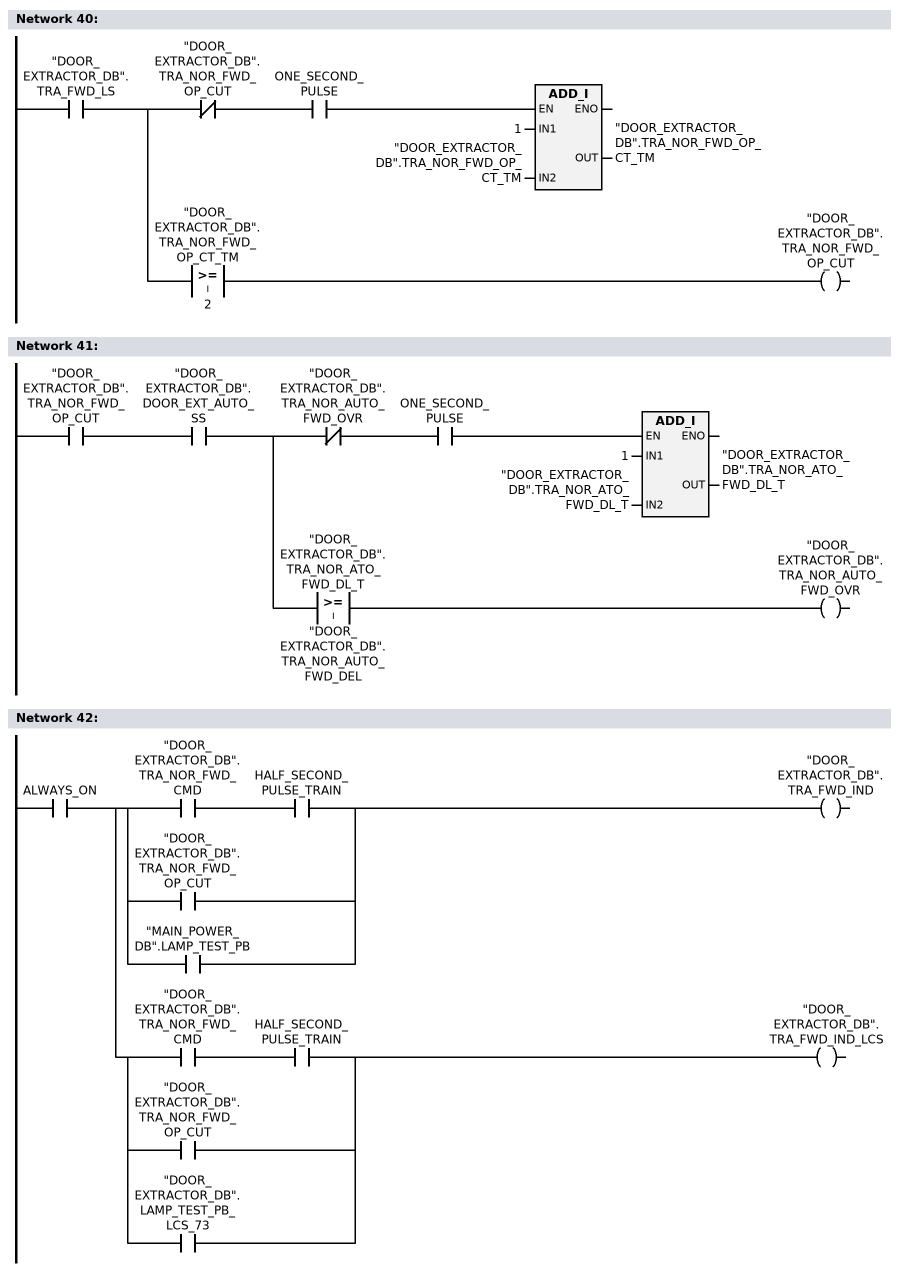
NETWORK
TITLE =
      A     "DOOR_EXTRACTOR_DB".TRA_FWD_LS;
      =     L 0.0;
      A     L 0.0;
      AN    "DOOR_EXTRACTOR_DB".TRA_NOR_FWD_OP_CUT;
      A     "ONE_SECOND_PULSE";
      JNB   M033;
      L     1;
      L     "DOOR_EXTRACTOR_DB".TRA_NOR_FWD_OP_CT_TM;
      +I;
      T     "DOOR_EXTRACTOR_DB".TRA_NOR_FWD_OP_CT_TM;
M033: NOP   0;
      A     L 0.0;
      A(;
      L     "DOOR_EXTRACTOR_DB".TRA_NOR_FWD_OP_CT_TM;
      L     2;
      >=I;
      );
      =     "DOOR_EXTRACTOR_DB".TRA_NOR_FWD_OP_CUT;
NETWORK
TITLE =
      A     "DOOR_EXTRACTOR_DB".TRA_NOR_FWD_OP_CUT;
      A     "DOOR_EXTRACTOR_DB".DOOR_EXT_AUTO_SS;
      =     L 0.0;
      A     L 0.0;
      AN    "DOOR_EXTRACTOR_DB".TRA_NOR_AUTO_FWD_OVR;
      A     "ONE_SECOND_PULSE";
      JNB   M034;
      L     1;
      L     "DOOR_EXTRACTOR_DB".TRA_NOR_ATO_FWD_DL_T;
      +I;
      T     "DOOR_EXTRACTOR_DB".TRA_NOR_ATO_FWD_DL_T;
M034: NOP   0;
      A     L 0.0;
      A(;
      L     "DOOR_EXTRACTOR_DB".TRA_NOR_ATO_FWD_DL_T;
      L     "DOOR_EXTRACTOR_DB".TRA_NOR_AUTO_FWD_DEL;
      >=I;
      );
      =     "DOOR_EXTRACTOR_DB".TRA_NOR_AUTO_FWD_OVR;
NETWORK
TITLE =
      A     "ALWAYS_ON";
      =     L 0.0;
      A     L 0.0;
      A(;
      A     "DOOR_EXTRACTOR_DB".TRA_NOR_FWD_CMD;
      A     "HALF_SECOND_PULSE_TRAIN";
      O     "DOOR_EXTRACTOR_DB".TRA_NOR_FWD_OP_CUT;
      O     "MAIN_POWER_DB".LAMP_TEST_PB;
      );
      =     "DOOR_EXTRACTOR_DB".TRA_FWD_IND;
      A     L 0.0;
      A(;
      A     "DOOR_EXTRACTOR_DB".TRA_NOR_FWD_CMD;
      A     "HALF_SECOND_PULSE_TRAIN";
      O     "DOOR_EXTRACTOR_DB".TRA_NOR_FWD_OP_CUT;
      O     "DOOR_EXTRACTOR_DB".LAMP_TEST_PB_LCS_73;
      );
      =     "DOOR_EXTRACTOR_DB".TRA_FWD_IND_LCS;
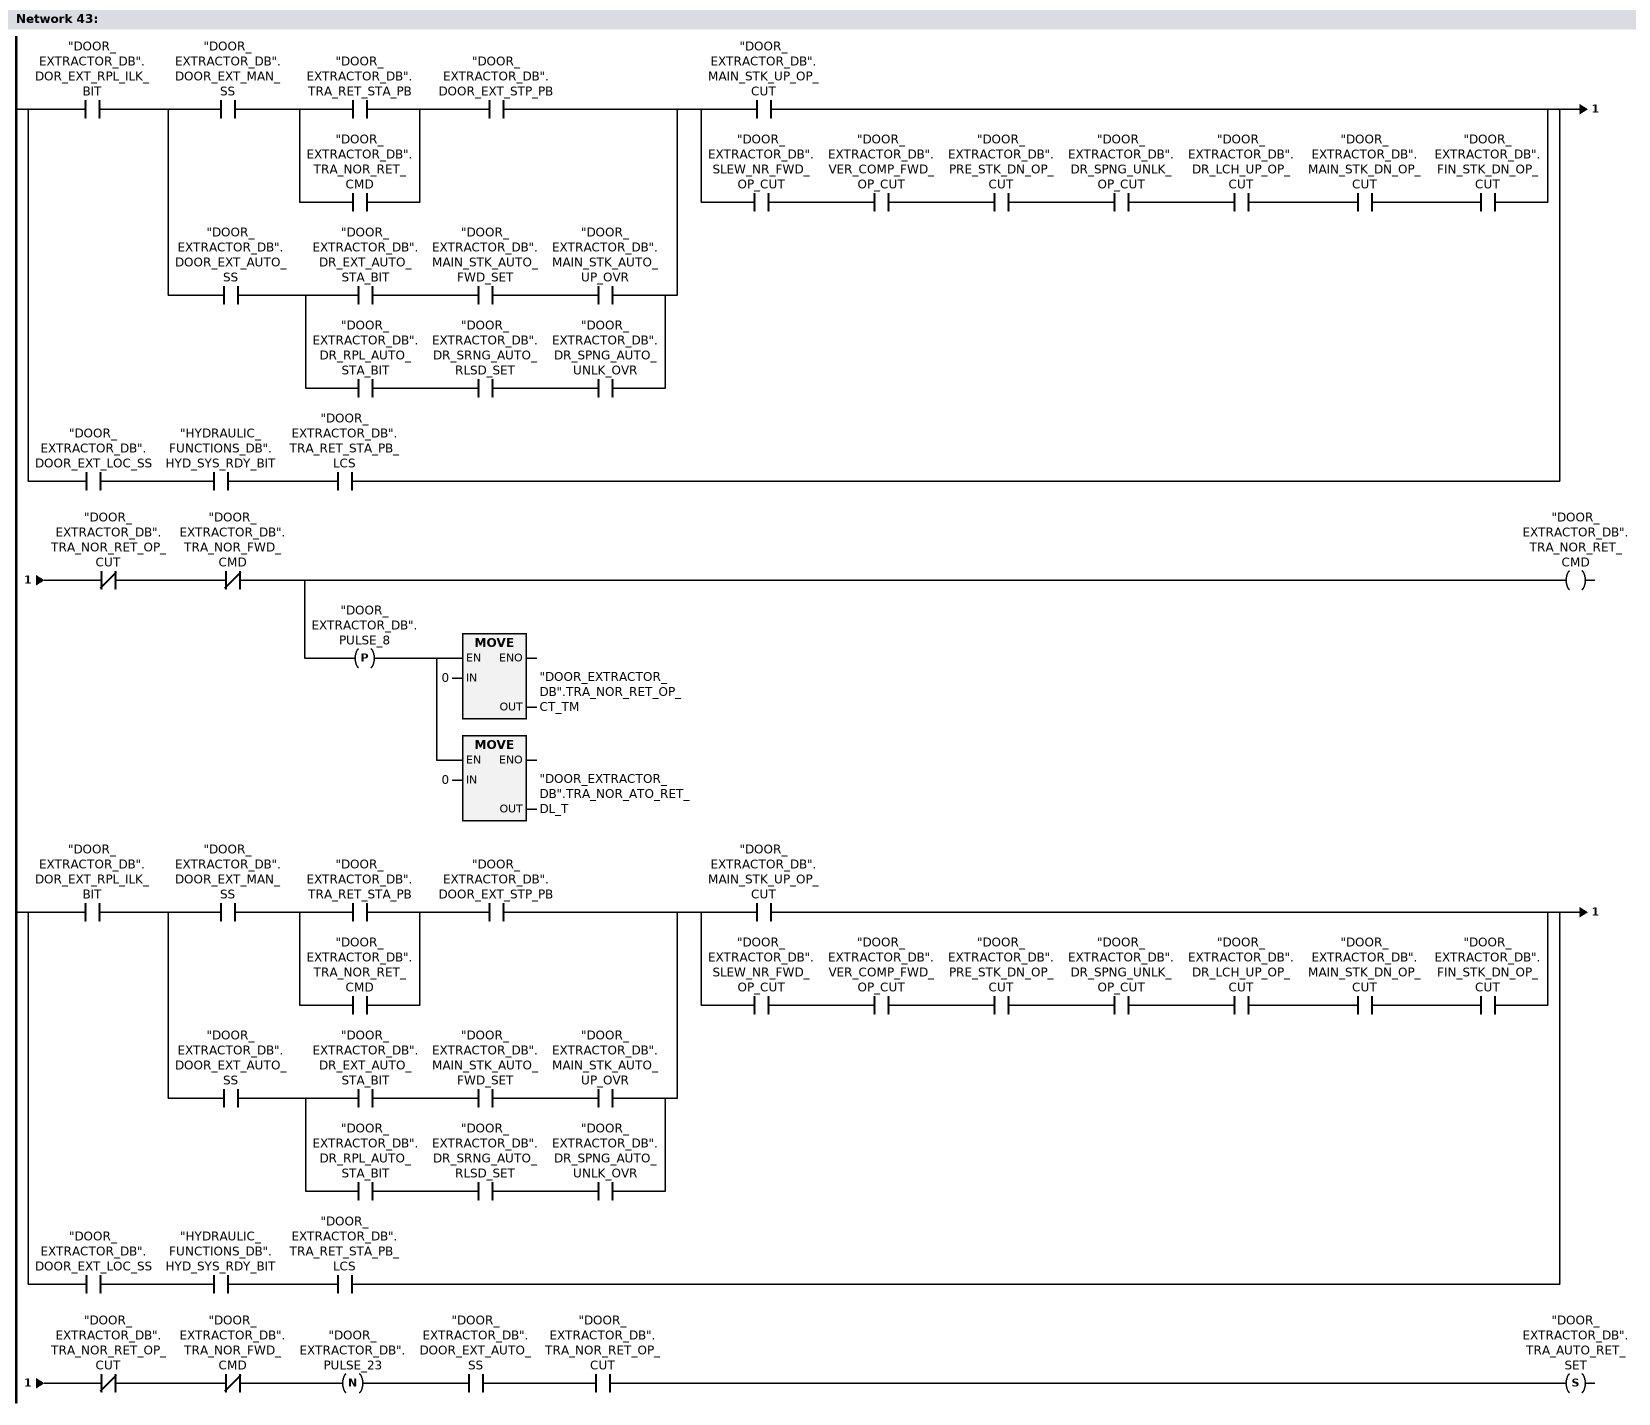
NETWORK
TITLE =
      A(;
      A     "DOOR_EXTRACTOR_DB".DOR_EXT_RPL_ILK_BIT;
      A(;
      A     "DOOR_EXTRACTOR_DB".DOOR_EXT_MAN_SS;
      A(;
      O     "DOOR_EXTRACTOR_DB".TRA_RET_STA_PB;
      O     "DOOR_EXTRACTOR_DB".TRA_NOR_RET_CMD;
      );
      A     "DOOR_EXTRACTOR_DB".DOOR_EXT_STP_PB;
      O;
      A     "DOOR_EXTRACTOR_DB".DOOR_EXT_AUTO_SS;
      A(;
      A     "DOOR_EXTRACTOR_DB".DR_EXT_AUTO_STA_BIT;
      A     "DOOR_EXTRACTOR_DB".MAIN_STK_AUTO_FWD_SET;
      A     "DOOR_EXTRACTOR_DB".MAIN_STK_AUTO_UP_OVR;
      O;
      A     "DOOR_EXTRACTOR_DB".DR_RPL_AUTO_STA_BIT;
      A     "DOOR_EXTRACTOR_DB".DR_SRNG_AUTO_RLSD_SET;
      A     "DOOR_EXTRACTOR_DB".DR_SPNG_AUTO_UNLK_OVR;
      );
      );
      A(;
      O     "DOOR_EXTRACTOR_DB".MAIN_STK_UP_OP_CUT;
      O;
      A     "DOOR_EXTRACTOR_DB".SLEW_NR_FWD_OP_CUT;
      A     "DOOR_EXTRACTOR_DB".VER_COMP_FWD_OP_CUT;
      A     "DOOR_EXTRACTOR_DB".PRE_STK_DN_OP_CUT;
      A     "DOOR_EXTRACTOR_DB".DR_SPNG_UNLK_OP_CUT;
      A     "DOOR_EXTRACTOR_DB".DR_LCH_UP_OP_CUT;
      A     "DOOR_EXTRACTOR_DB".MAIN_STK_DN_OP_CUT;
      A     "DOOR_EXTRACTOR_DB".FIN_STK_DN_OP_CUT;
      );
      O;
      A     "DOOR_EXTRACTOR_DB".DOOR_EXT_LOC_SS;
      A     "HYDRAULIC_FUNCTIONS_DB".HYD_SYS_RDY_BIT;
      A     "DOOR_EXTRACTOR_DB".TRA_RET_STA_PB_LCS;
      );
      AN    "DOOR_EXTRACTOR_DB".TRA_NOR_RET_OP_CUT;
      AN    "DOOR_EXTRACTOR_DB".TRA_NOR_FWD_CMD;
      =     L 0.0;
      A     L 0.0;
      BLD   102;
      =     "DOOR_EXTRACTOR_DB".TRA_NOR_RET_CMD;
      A(;
      A     L 0.0;
      FN    "DOOR_EXTRACTOR_DB".PULSE_23;
      );
      A     "DOOR_EXTRACTOR_DB".DOOR_EXT_AUTO_SS;
      A     "DOOR_EXTRACTOR_DB".TRA_NOR_RET_OP_CUT;
      S     "DOOR_EXTRACTOR_DB".TRA_AUTO_RET_SET;
      A     L 0.0;
      FP    "DOOR_EXTRACTOR_DB".PULSE_8;
      =     L 0.1;
      A     L 0.1;
      JNB   M035;
      L     0;
      T     "DOOR_EXTRACTOR_DB".TRA_NOR_RET_OP_CT_TM;
M035: NOP   0;
      A     L 0.1;
      JNB   M036;
      L     0;
      T     "DOOR_EXTRACTOR_DB".TRA_NOR_ATO_RET_DL_T;
M036: NOP   0;
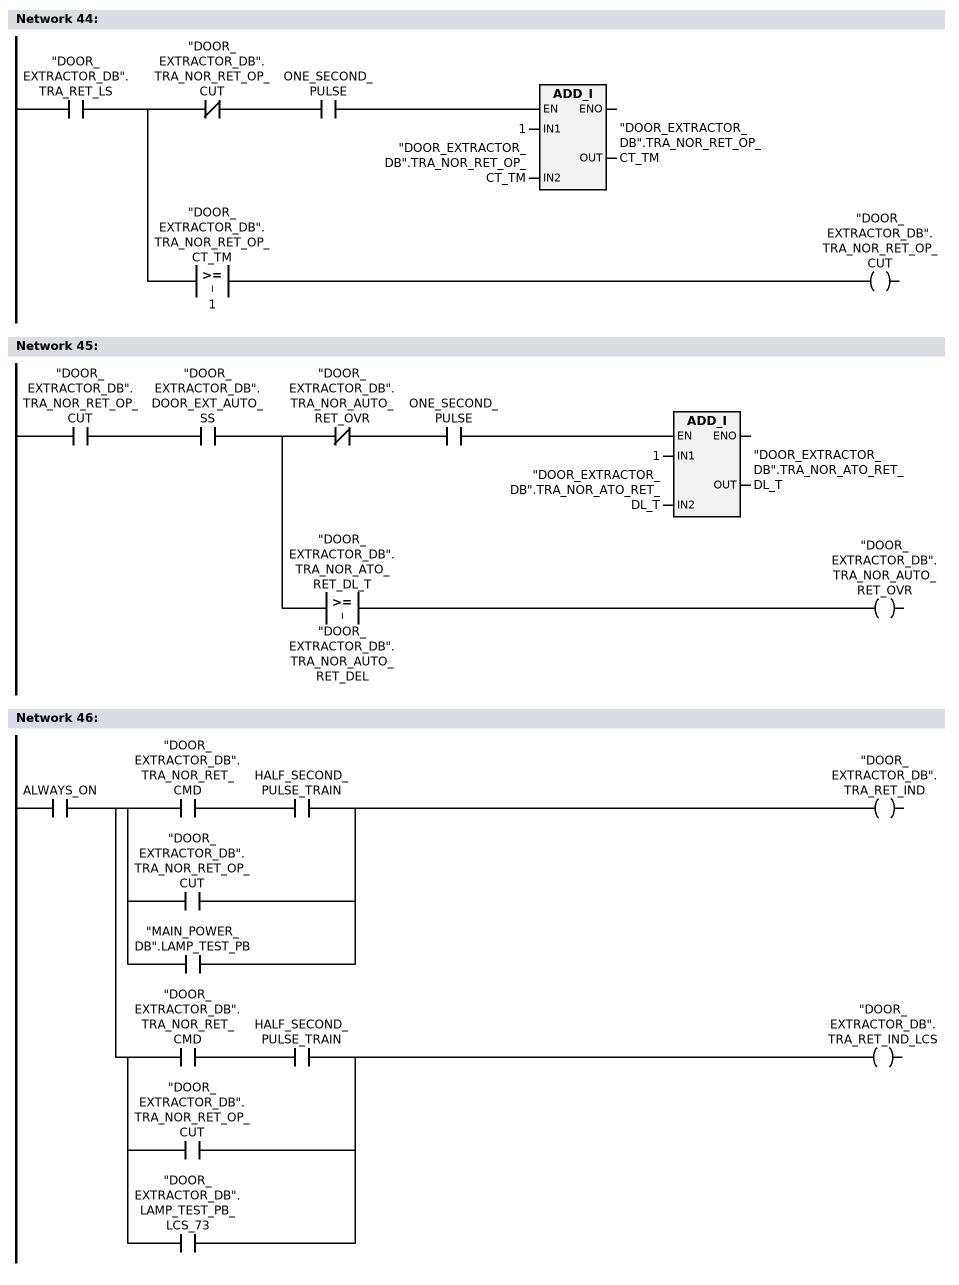
NETWORK
TITLE =
      A     "DOOR_EXTRACTOR_DB".TRA_RET_LS;
      =     L 0.0;
      A     L 0.0;
      AN    "DOOR_EXTRACTOR_DB".TRA_NOR_RET_OP_CUT;
      A     "ONE_SECOND_PULSE";
      JNB   M037;
      L     1;
      L     "DOOR_EXTRACTOR_DB".TRA_NOR_RET_OP_CT_TM;
      +I;
      T     "DOOR_EXTRACTOR_DB".TRA_NOR_RET_OP_CT_TM;
M037: NOP   0;
      A     L 0.0;
      A(;
      L     "DOOR_EXTRACTOR_DB".TRA_NOR_RET_OP_CT_TM;
      L     1;
      >=I;
      );
      =     "DOOR_EXTRACTOR_DB".TRA_NOR_RET_OP_CUT;
NETWORK
TITLE =
      A     "DOOR_EXTRACTOR_DB".TRA_NOR_RET_OP_CUT;
      A     "DOOR_EXTRACTOR_DB".DOOR_EXT_AUTO_SS;
      =     L 0.0;
      A     L 0.0;
      AN    "DOOR_EXTRACTOR_DB".TRA_NOR_AUTO_RET_OVR;
      A     "ONE_SECOND_PULSE";
      JNB   M038;
      L     1;
      L     "DOOR_EXTRACTOR_DB".TRA_NOR_ATO_RET_DL_T;
      +I;
      T     "DOOR_EXTRACTOR_DB".TRA_NOR_ATO_RET_DL_T;
M038: NOP   0;
      A     L 0.0;
      A(;
      L     "DOOR_EXTRACTOR_DB".TRA_NOR_ATO_RET_DL_T;
      L     "DOOR_EXTRACTOR_DB".TRA_NOR_AUTO_RET_DEL;
      >=I;
      );
      =     "DOOR_EXTRACTOR_DB".TRA_NOR_AUTO_RET_OVR;
NETWORK
TITLE =
      A     "ALWAYS_ON";
      =     L 0.0;
      A     L 0.0;
      A(;
      A     "DOOR_EXTRACTOR_DB".TRA_NOR_RET_CMD;
      A     "HALF_SECOND_PULSE_TRAIN";
      O     "DOOR_EXTRACTOR_DB".TRA_NOR_RET_OP_CUT;
      O     "MAIN_POWER_DB".LAMP_TEST_PB;
      );
      =     "DOOR_EXTRACTOR_DB".TRA_RET_IND;
      A     L 0.0;
      A(;
      A     "DOOR_EXTRACTOR_DB".TRA_NOR_RET_CMD;
      A     "HALF_SECOND_PULSE_TRAIN";
      O     "DOOR_EXTRACTOR_DB".TRA_NOR_RET_OP_CUT;
      O     "DOOR_EXTRACTOR_DB".LAMP_TEST_PB_LCS_73;
      );
      =     "DOOR_EXTRACTOR_DB".TRA_RET_IND_LCS;
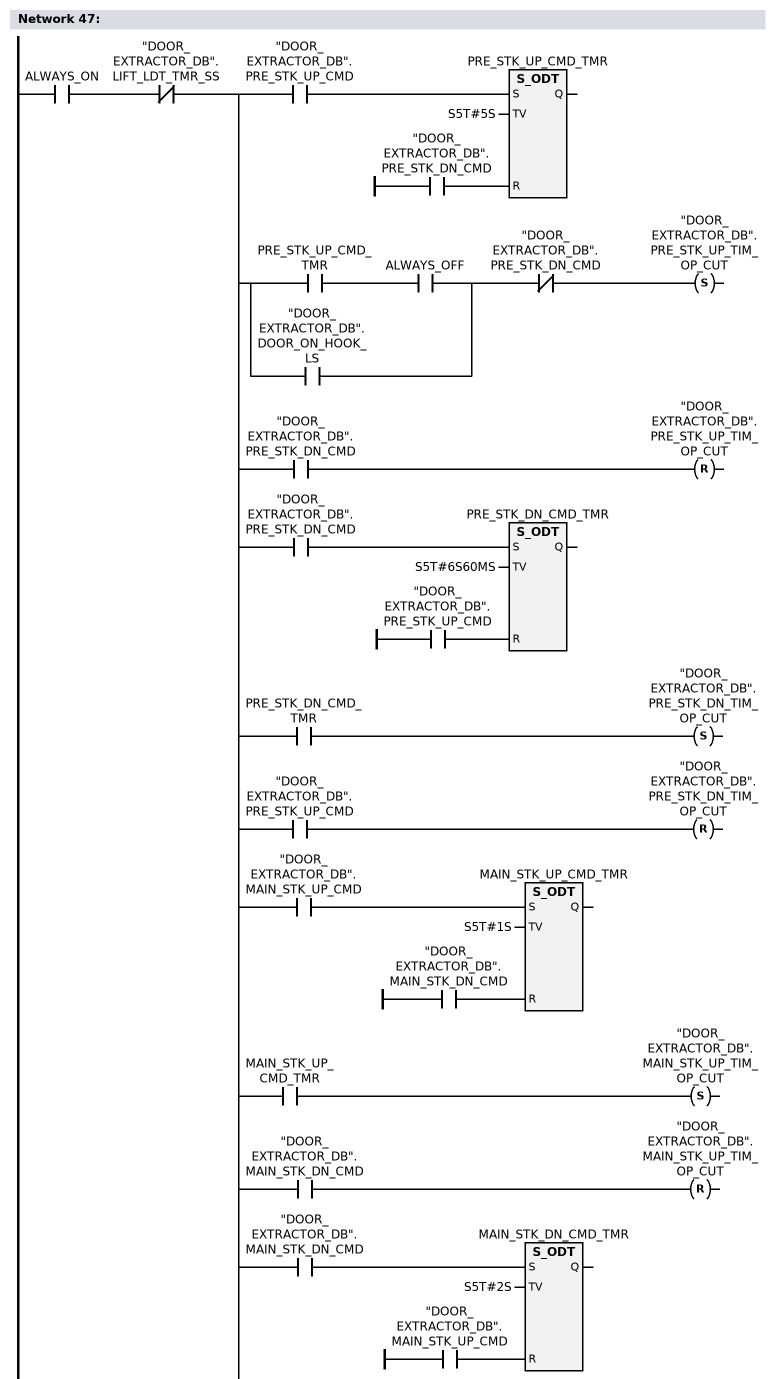
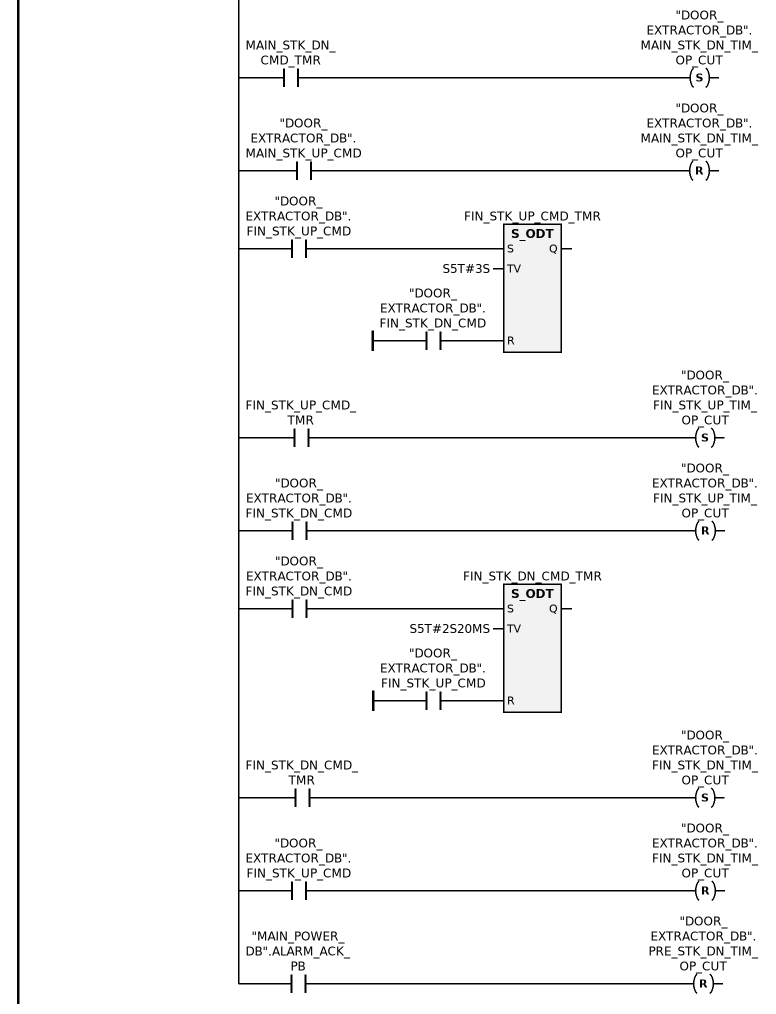
NETWORK
TITLE =
      A     "ALWAYS_ON";
      AN    "DOOR_EXTRACTOR_DB".LIFT_LDT_TMR_SS;
      =     L 0.0;
      A     L 0.0;
      A     "DOOR_EXTRACTOR_DB".PRE_STK_UP_CMD;
      L     S5T#5S;
      SD    "PRE_STK_UP_CMD_TMR";
      A     "DOOR_EXTRACTOR_DB".PRE_STK_DN_CMD;
      R     "PRE_STK_UP_CMD_TMR";
      NOP   0;
      NOP   0;
      NOP   0;
      A     L 0.0;
      A(;
      A     "PRE_STK_UP_CMD_TMR";
      A     "ALWAYS_OFF";
      O     "DOOR_EXTRACTOR_DB".DOOR_ON_HOOK_LS;
      );
      AN    "DOOR_EXTRACTOR_DB".PRE_STK_DN_CMD;
      S     "DOOR_EXTRACTOR_DB".PRE_STK_UP_TIM_OP_CUT;
      A     L 0.0;
      A     "DOOR_EXTRACTOR_DB".PRE_STK_DN_CMD;
      R     "DOOR_EXTRACTOR_DB".PRE_STK_UP_TIM_OP_CUT;
      A     L 0.0;
      A     "DOOR_EXTRACTOR_DB".PRE_STK_DN_CMD;
      L     S5T#6S60MS;
      SD    "PRE_STK_DN_CMD_TMR";
      A     "DOOR_EXTRACTOR_DB".PRE_STK_UP_CMD;
      R     "PRE_STK_DN_CMD_TMR";
      NOP   0;
      NOP   0;
      NOP   0;
      A     L 0.0;
      A     "PRE_STK_DN_CMD_TMR";
      S     "DOOR_EXTRACTOR_DB".PRE_STK_DN_TIM_OP_CUT;
      A     L 0.0;
      A     "DOOR_EXTRACTOR_DB".PRE_STK_UP_CMD;
      R     "DOOR_EXTRACTOR_DB".PRE_STK_DN_TIM_OP_CUT;
      A     L 0.0;
      A     "DOOR_EXTRACTOR_DB".MAIN_STK_UP_CMD;
      L     S5T#1S;
      SD    "MAIN_STK_UP_CMD_TMR";
      A     "DOOR_EXTRACTOR_DB".MAIN_STK_DN_CMD;
      R     "MAIN_STK_UP_CMD_TMR";
      NOP   0;
      NOP   0;
      NOP   0;
      A     L 0.0;
      A     "MAIN_STK_UP_CMD_TMR";
      S     "DOOR_EXTRACTOR_DB".MAIN_STK_UP_TIM_OP_CUT;
      A     L 0.0;
      A     "DOOR_EXTRACTOR_DB".MAIN_STK_DN_CMD;
      R     "DOOR_EXTRACTOR_DB".MAIN_STK_UP_TIM_OP_CUT;
      A     L 0.0;
      A     "DOOR_EXTRACTOR_DB".MAIN_STK_DN_CMD;
      L     S5T#2S;
      SD    "MAIN_STK_DN_CMD_TMR";
      A     "DOOR_EXTRACTOR_DB".MAIN_STK_UP_CMD;
      R     "MAIN_STK_DN_CMD_TMR";
      NOP   0;
      NOP   0;
      NOP   0;
      A     L 0.0;
      A     "MAIN_STK_DN_CMD_TMR";
      S     "DOOR_EXTRACTOR_DB".MAIN_STK_DN_TIM_OP_CUT;
      A     L 0.0;
      A     "DOOR_EXTRACTOR_DB".MAIN_STK_UP_CMD;
      R     "DOOR_EXTRACTOR_DB".MAIN_STK_DN_TIM_OP_CUT;
      A     L 0.0;
      A     "DOOR_EXTRACTOR_DB".FIN_STK_UP_CMD;
      L     S5T#3S;
      SD    "FIN_STK_UP_CMD_TMR";
      A     "DOOR_EXTRACTOR_DB".FIN_STK_DN_CMD;
      R     "FIN_STK_UP_CMD_TMR";
      NOP   0;
      NOP   0;
      NOP   0;
      A     L 0.0;
      A     "FIN_STK_UP_CMD_TMR";
      S     "DOOR_EXTRACTOR_DB".FIN_STK_UP_TIM_OP_CUT;
      A     L 0.0;
      A     "DOOR_EXTRACTOR_DB".FIN_STK_DN_CMD;
      R     "DOOR_EXTRACTOR_DB".FIN_STK_UP_TIM_OP_CUT;
      A     L 0.0;
      A     "DOOR_EXTRACTOR_DB".FIN_STK_DN_CMD;
      L     S5T#2S20MS;
      SD    "FIN_STK_DN_CMD_TMR";
      A     "DOOR_EXTRACTOR_DB".FIN_STK_UP_CMD;
      R     "FIN_STK_DN_CMD_TMR";
      NOP   0;
      NOP   0;
      NOP   0;
      A     L 0.0;
      A     "FIN_STK_DN_CMD_TMR";
      S     "DOOR_EXTRACTOR_DB".FIN_STK_DN_TIM_OP_CUT;
      A     L 0.0;
      A     "DOOR_EXTRACTOR_DB".FIN_STK_UP_CMD;
      R     "DOOR_EXTRACTOR_DB".FIN_STK_DN_TIM_OP_CUT;
      A     L 0.0;
      A     "MAIN_POWER_DB".ALARM_ACK_PB;
      R     "DOOR_EXTRACTOR_DB".PRE_STK_DN_TIM_OP_CUT;
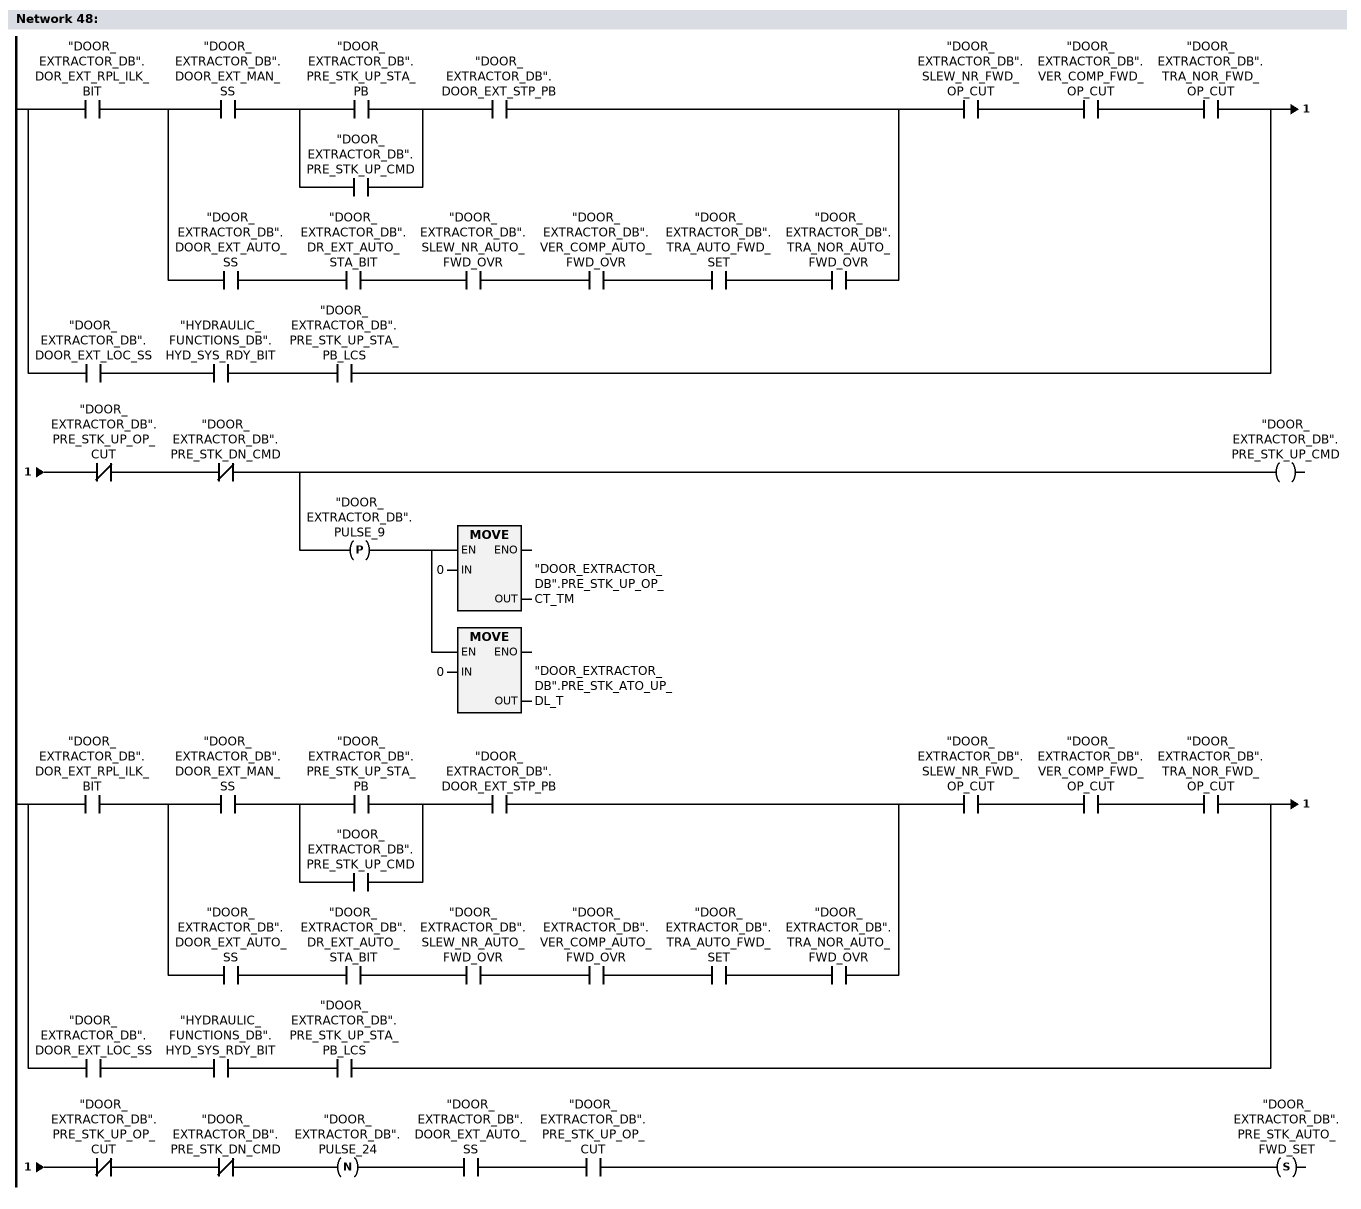
NETWORK
TITLE =
      A(;
      A     "DOOR_EXTRACTOR_DB".DOR_EXT_RPL_ILK_BIT;
      A(;
      A     "DOOR_EXTRACTOR_DB".DOOR_EXT_MAN_SS;
      A(;
      O     "DOOR_EXTRACTOR_DB".PRE_STK_UP_STA_PB;
      O     "DOOR_EXTRACTOR_DB".PRE_STK_UP_CMD;
      );
      A     "DOOR_EXTRACTOR_DB".DOOR_EXT_STP_PB;
      O;
      A     "DOOR_EXTRACTOR_DB".DOOR_EXT_AUTO_SS;
      A     "DOOR_EXTRACTOR_DB".DR_EXT_AUTO_STA_BIT;
      A     "DOOR_EXTRACTOR_DB".SLEW_NR_AUTO_FWD_OVR;
      A     "DOOR_EXTRACTOR_DB".VER_COMP_AUTO_FWD_OVR;
      A     "DOOR_EXTRACTOR_DB".TRA_AUTO_FWD_SET;
      A     "DOOR_EXTRACTOR_DB".TRA_NOR_AUTO_FWD_OVR;
      );
      A     "DOOR_EXTRACTOR_DB".SLEW_NR_FWD_OP_CUT;
      A     "DOOR_EXTRACTOR_DB".VER_COMP_FWD_OP_CUT;
      A     "DOOR_EXTRACTOR_DB".TRA_NOR_FWD_OP_CUT;
      O;
      A     "DOOR_EXTRACTOR_DB".DOOR_EXT_LOC_SS;
      A     "HYDRAULIC_FUNCTIONS_DB".HYD_SYS_RDY_BIT;
      A     "DOOR_EXTRACTOR_DB".PRE_STK_UP_STA_PB_LCS;
      );
      AN    "DOOR_EXTRACTOR_DB".PRE_STK_UP_OP_CUT;
      AN    "DOOR_EXTRACTOR_DB".PRE_STK_DN_CMD;
      =     L 0.0;
      A     L 0.0;
      BLD   102;
      =     "DOOR_EXTRACTOR_DB".PRE_STK_UP_CMD;
      A(;
      A     L 0.0;
      FN    "DOOR_EXTRACTOR_DB".PULSE_24;
      );
      A     "DOOR_EXTRACTOR_DB".DOOR_EXT_AUTO_SS;
      A     "DOOR_EXTRACTOR_DB".PRE_STK_UP_OP_CUT;
      S     "DOOR_EXTRACTOR_DB".PRE_STK_AUTO_FWD_SET;
      A     L 0.0;
      FP    "DOOR_EXTRACTOR_DB".PULSE_9;
      =     L 0.1;
      A     L 0.1;
      JNB   M039;
      L     0;
      T     "DOOR_EXTRACTOR_DB".PRE_STK_UP_OP_CT_TM;
M039: NOP   0;
      A     L 0.1;
      JNB   M040;
      L     0;
      T     "DOOR_EXTRACTOR_DB".PRE_STK_ATO_UP_DL_T;
M040: NOP   0;
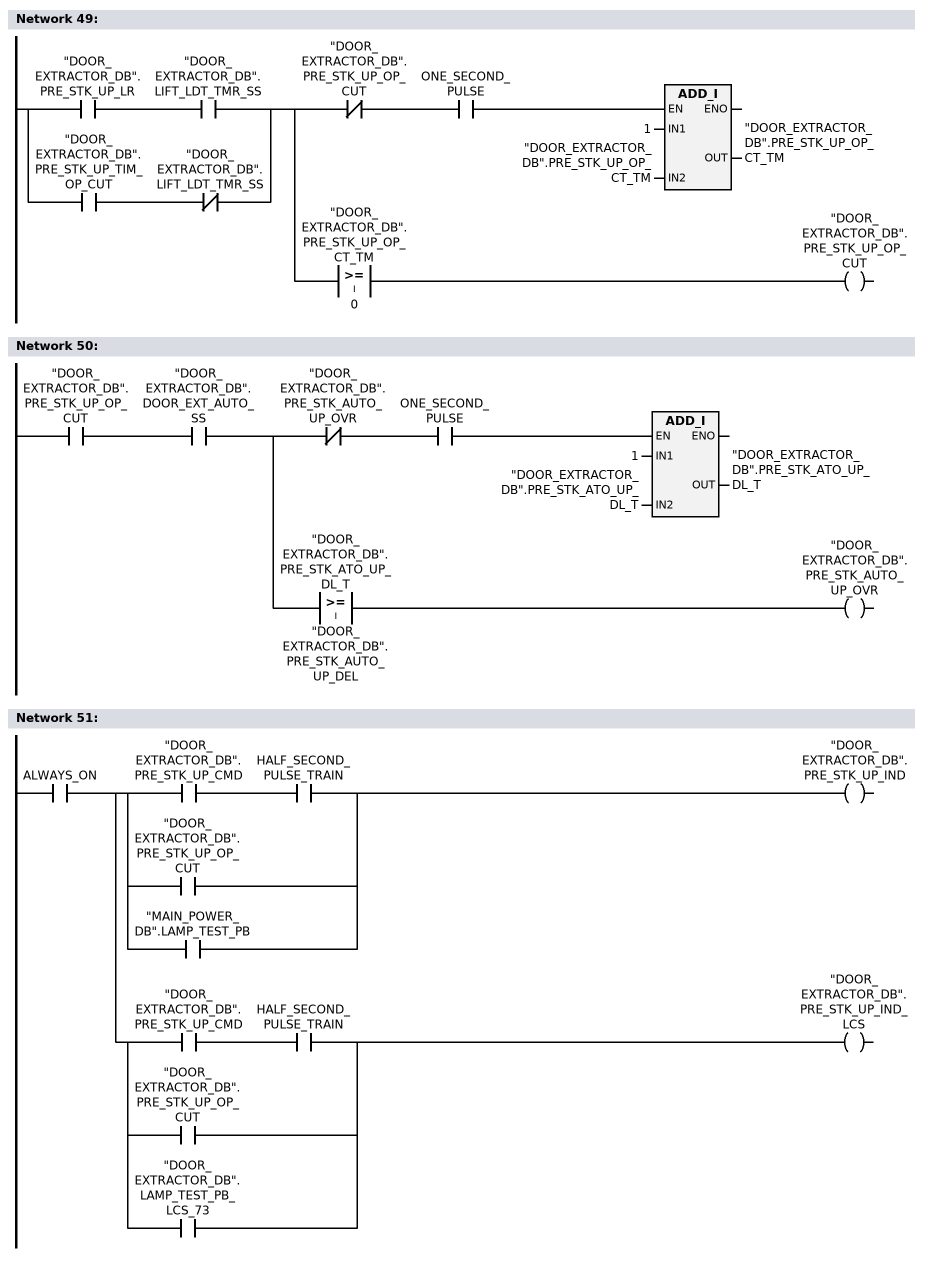
NETWORK
TITLE =
      A     "DOOR_EXTRACTOR_DB".PRE_STK_UP_LR;
      A     "DOOR_EXTRACTOR_DB".LIFT_LDT_TMR_SS;
      O;
      A     "DOOR_EXTRACTOR_DB".PRE_STK_UP_TIM_OP_CUT;
      AN    "DOOR_EXTRACTOR_DB".LIFT_LDT_TMR_SS;
      =     L 0.0;
      A     L 0.0;
      AN    "DOOR_EXTRACTOR_DB".PRE_STK_UP_OP_CUT;
      A     "ONE_SECOND_PULSE";
      JNB   M041;
      L     1;
      L     "DOOR_EXTRACTOR_DB".PRE_STK_UP_OP_CT_TM;
      +I;
      T     "DOOR_EXTRACTOR_DB".PRE_STK_UP_OP_CT_TM;
M041: NOP   0;
      A     L 0.0;
      A(;
      L     "DOOR_EXTRACTOR_DB".PRE_STK_UP_OP_CT_TM;
      L     0;
      >=I;
      );
      =     "DOOR_EXTRACTOR_DB".PRE_STK_UP_OP_CUT;
NETWORK
TITLE =
      A     "DOOR_EXTRACTOR_DB".PRE_STK_UP_OP_CUT;
      A     "DOOR_EXTRACTOR_DB".DOOR_EXT_AUTO_SS;
      =     L 0.0;
      A     L 0.0;
      AN    "DOOR_EXTRACTOR_DB".PRE_STK_AUTO_UP_OVR;
      A     "ONE_SECOND_PULSE";
      JNB   M042;
      L     1;
      L     "DOOR_EXTRACTOR_DB".PRE_STK_ATO_UP_DL_T;
      +I;
      T     "DOOR_EXTRACTOR_DB".PRE_STK_ATO_UP_DL_T;
M042: NOP   0;
      A     L 0.0;
      A(;
      L     "DOOR_EXTRACTOR_DB".PRE_STK_ATO_UP_DL_T;
      L     "DOOR_EXTRACTOR_DB".PRE_STK_AUTO_UP_DEL;
      >=I;
      );
      =     "DOOR_EXTRACTOR_DB".PRE_STK_AUTO_UP_OVR;
NETWORK
TITLE =
      A     "ALWAYS_ON";
      =     L 0.0;
      A     L 0.0;
      A(;
      A     "DOOR_EXTRACTOR_DB".PRE_STK_UP_CMD;
      A     "HALF_SECOND_PULSE_TRAIN";
      O     "DOOR_EXTRACTOR_DB".PRE_STK_UP_OP_CUT;
      O     "MAIN_POWER_DB".LAMP_TEST_PB;
      );
      =     "DOOR_EXTRACTOR_DB".PRE_STK_UP_IND;
      A     L 0.0;
      A(;
      A     "DOOR_EXTRACTOR_DB".PRE_STK_UP_CMD;
      A     "HALF_SECOND_PULSE_TRAIN";
      O     "DOOR_EXTRACTOR_DB".PRE_STK_UP_OP_CUT;
      O     "DOOR_EXTRACTOR_DB".LAMP_TEST_PB_LCS_73;
      );
      =     "DOOR_EXTRACTOR_DB".PRE_STK_UP_IND_LCS;
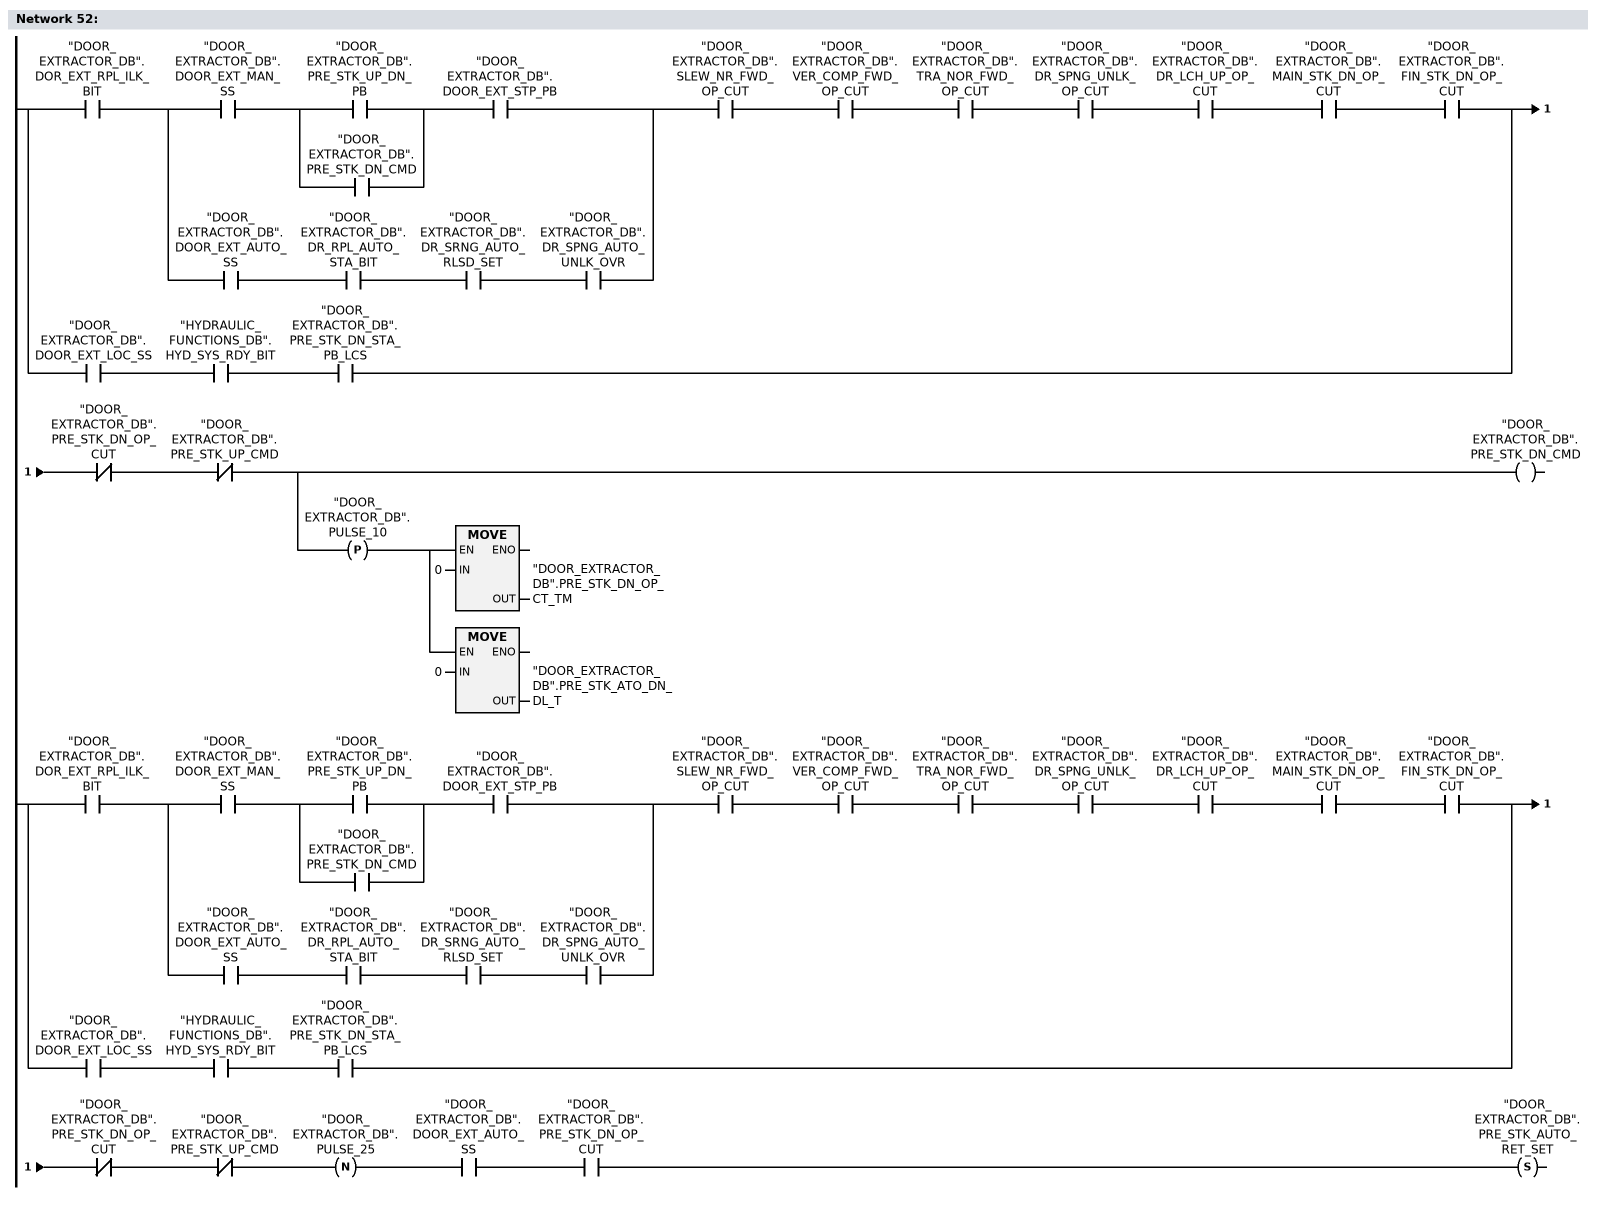
NETWORK
TITLE =
      A(;
      A     "DOOR_EXTRACTOR_DB".DOR_EXT_RPL_ILK_BIT;
      A(;
      A     "DOOR_EXTRACTOR_DB".DOOR_EXT_MAN_SS;
      A(;
      O     "DOOR_EXTRACTOR_DB".PRE_STK_UP_DN_PB;
      O     "DOOR_EXTRACTOR_DB".PRE_STK_DN_CMD;
      );
      A     "DOOR_EXTRACTOR_DB".DOOR_EXT_STP_PB;
      O;
      A     "DOOR_EXTRACTOR_DB".DOOR_EXT_AUTO_SS;
      A     "DOOR_EXTRACTOR_DB".DR_RPL_AUTO_STA_BIT;
      A     "DOOR_EXTRACTOR_DB".DR_SRNG_AUTO_RLSD_SET;
      A     "DOOR_EXTRACTOR_DB".DR_SPNG_AUTO_UNLK_OVR;
      );
      A     "DOOR_EXTRACTOR_DB".SLEW_NR_FWD_OP_CUT;
      A     "DOOR_EXTRACTOR_DB".VER_COMP_FWD_OP_CUT;
      A     "DOOR_EXTRACTOR_DB".TRA_NOR_FWD_OP_CUT;
      A     "DOOR_EXTRACTOR_DB".DR_SPNG_UNLK_OP_CUT;
      A     "DOOR_EXTRACTOR_DB".DR_LCH_UP_OP_CUT;
      A     "DOOR_EXTRACTOR_DB".MAIN_STK_DN_OP_CUT;
      A     "DOOR_EXTRACTOR_DB".FIN_STK_DN_OP_CUT;
      O;
      A     "DOOR_EXTRACTOR_DB".DOOR_EXT_LOC_SS;
      A     "HYDRAULIC_FUNCTIONS_DB".HYD_SYS_RDY_BIT;
      A     "DOOR_EXTRACTOR_DB".PRE_STK_DN_STA_PB_LCS;
      );
      AN    "DOOR_EXTRACTOR_DB".PRE_STK_DN_OP_CUT;
      AN    "DOOR_EXTRACTOR_DB".PRE_STK_UP_CMD;
      =     L 0.0;
      A     L 0.0;
      BLD   102;
      =     "DOOR_EXTRACTOR_DB".PRE_STK_DN_CMD;
      A(;
      A     L 0.0;
      FN    "DOOR_EXTRACTOR_DB".PULSE_25;
      );
      A     "DOOR_EXTRACTOR_DB".DOOR_EXT_AUTO_SS;
      A     "DOOR_EXTRACTOR_DB".PRE_STK_DN_OP_CUT;
      S     "DOOR_EXTRACTOR_DB".PRE_STK_AUTO_RET_SET;
      A     L 0.0;
      FP    "DOOR_EXTRACTOR_DB".PULSE_10;
      =     L 0.1;
      A     L 0.1;
      JNB   M043;
      L     0;
      T     "DOOR_EXTRACTOR_DB".PRE_STK_DN_OP_CT_TM;
M043: NOP   0;
      A     L 0.1;
      JNB   M044;
      L     0;
      T     "DOOR_EXTRACTOR_DB".PRE_STK_ATO_DN_DL_T;
M044: NOP   0;
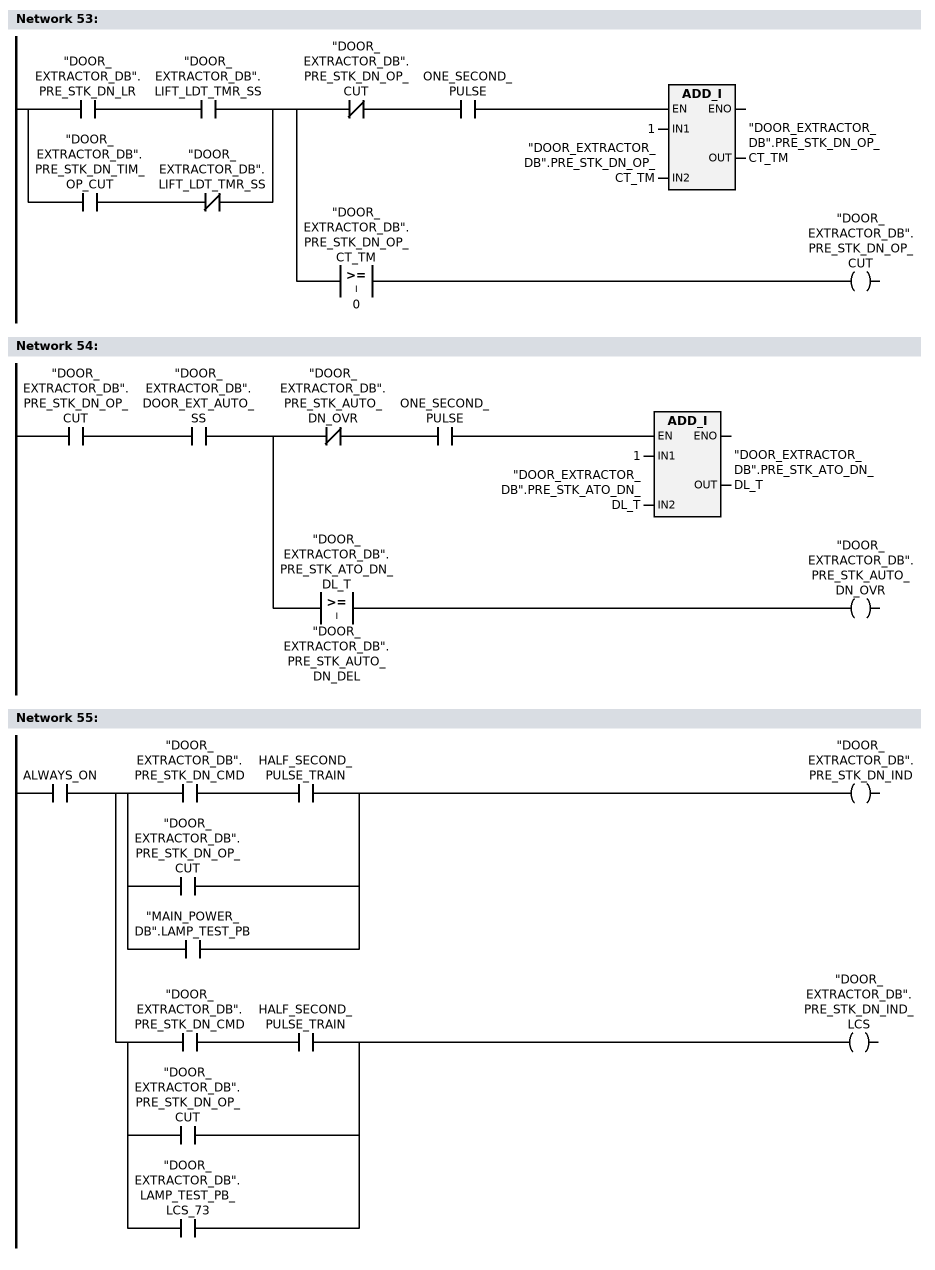
NETWORK
TITLE =
      A     "DOOR_EXTRACTOR_DB".PRE_STK_DN_LR;
      A     "DOOR_EXTRACTOR_DB".LIFT_LDT_TMR_SS;
      O;
      A     "DOOR_EXTRACTOR_DB".PRE_STK_DN_TIM_OP_CUT;
      AN    "DOOR_EXTRACTOR_DB".LIFT_LDT_TMR_SS;
      =     L 0.0;
      A     L 0.0;
      AN    "DOOR_EXTRACTOR_DB".PRE_STK_DN_OP_CUT;
      A     "ONE_SECOND_PULSE";
      JNB   M045;
      L     1;
      L     "DOOR_EXTRACTOR_DB".PRE_STK_DN_OP_CT_TM;
      +I;
      T     "DOOR_EXTRACTOR_DB".PRE_STK_DN_OP_CT_TM;
M045: NOP   0;
      A     L 0.0;
      A(;
      L     "DOOR_EXTRACTOR_DB".PRE_STK_DN_OP_CT_TM;
      L     0;
      >=I;
      );
      =     "DOOR_EXTRACTOR_DB".PRE_STK_DN_OP_CUT;
NETWORK
TITLE =
      A     "DOOR_EXTRACTOR_DB".PRE_STK_DN_OP_CUT;
      A     "DOOR_EXTRACTOR_DB".DOOR_EXT_AUTO_SS;
      =     L 0.0;
      A     L 0.0;
      AN    "DOOR_EXTRACTOR_DB".PRE_STK_AUTO_DN_OVR;
      A     "ONE_SECOND_PULSE";
      JNB   M046;
      L     1;
      L     "DOOR_EXTRACTOR_DB".PRE_STK_ATO_DN_DL_T;
      +I;
      T     "DOOR_EXTRACTOR_DB".PRE_STK_ATO_DN_DL_T;
M046: NOP   0;
      A     L 0.0;
      A(;
      L     "DOOR_EXTRACTOR_DB".PRE_STK_ATO_DN_DL_T;
      L     "DOOR_EXTRACTOR_DB".PRE_STK_AUTO_DN_DEL;
      >=I;
      );
      =     "DOOR_EXTRACTOR_DB".PRE_STK_AUTO_DN_OVR;
NETWORK
TITLE =
      A     "ALWAYS_ON";
      =     L 0.0;
      A     L 0.0;
      A(;
      A     "DOOR_EXTRACTOR_DB".PRE_STK_DN_CMD;
      A     "HALF_SECOND_PULSE_TRAIN";
      O     "DOOR_EXTRACTOR_DB".PRE_STK_DN_OP_CUT;
      O     "MAIN_POWER_DB".LAMP_TEST_PB;
      );
      =     "DOOR_EXTRACTOR_DB".PRE_STK_DN_IND;
      A     L 0.0;
      A(;
      A     "DOOR_EXTRACTOR_DB".PRE_STK_DN_CMD;
      A     "HALF_SECOND_PULSE_TRAIN";
      O     "DOOR_EXTRACTOR_DB".PRE_STK_DN_OP_CUT;
      O     "DOOR_EXTRACTOR_DB".LAMP_TEST_PB_LCS_73;
      );
      =     "DOOR_EXTRACTOR_DB".PRE_STK_DN_IND_LCS;
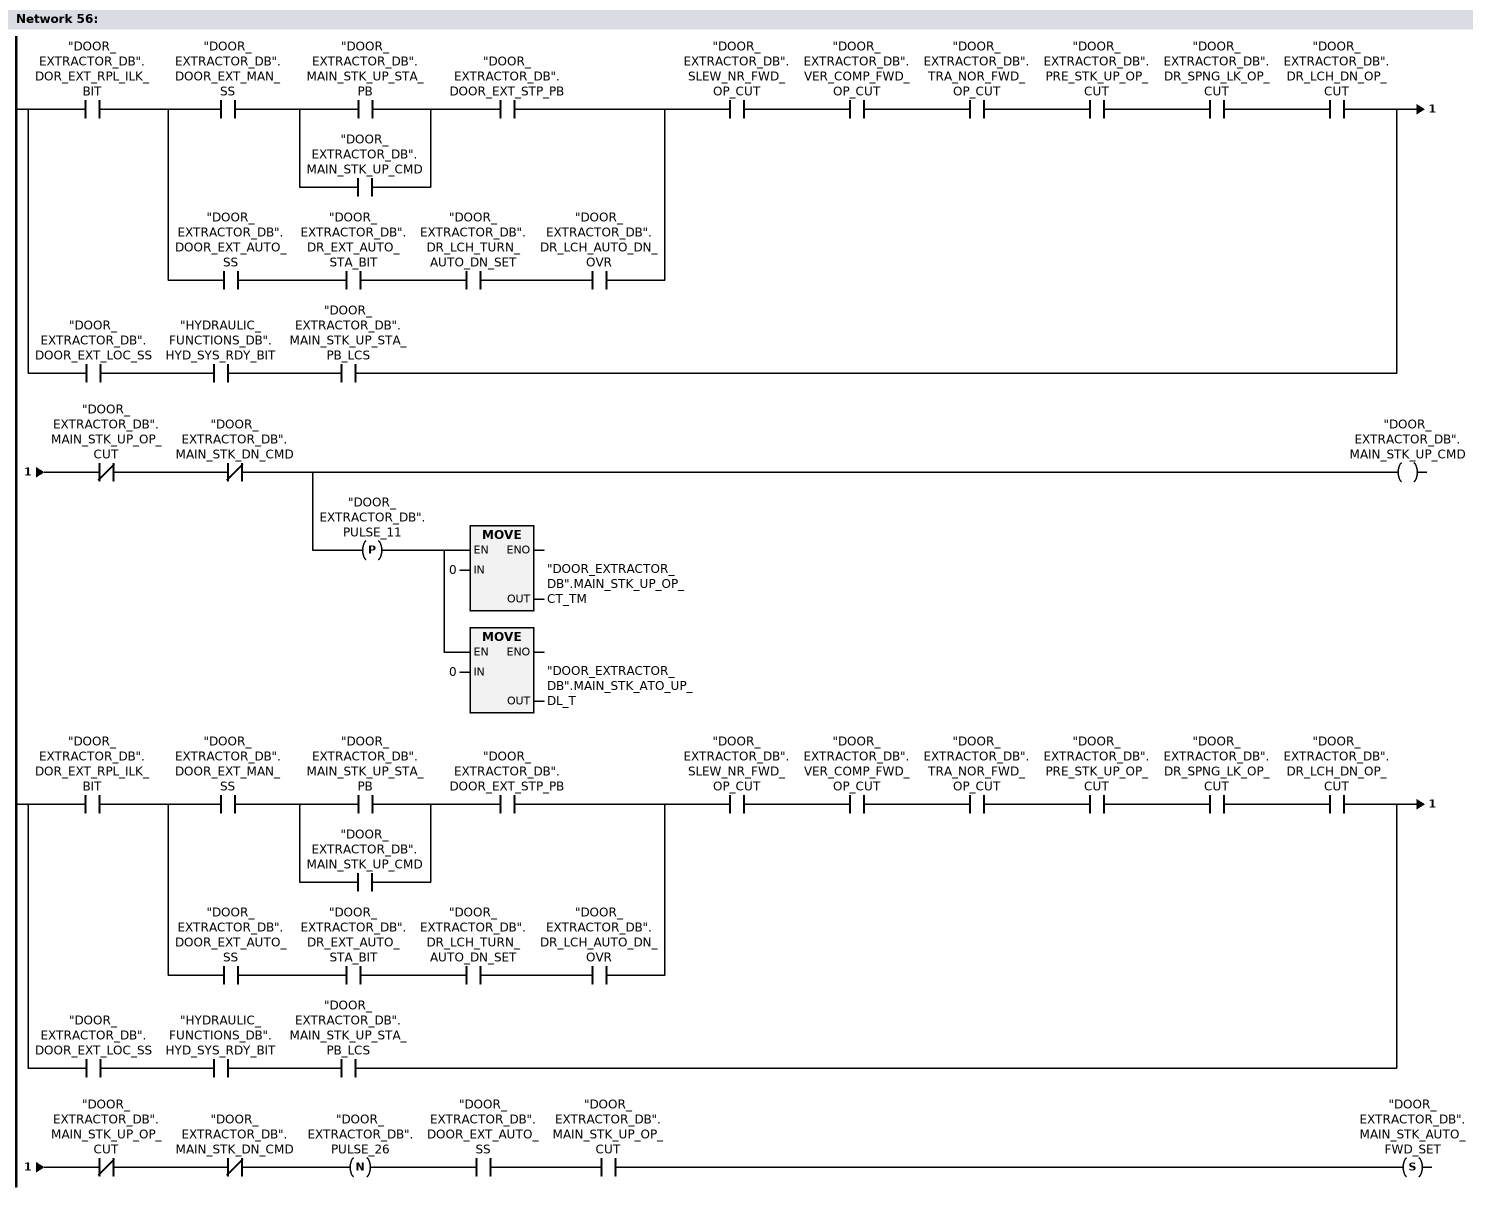
NETWORK
TITLE =
      A(;
      A     "DOOR_EXTRACTOR_DB".DOR_EXT_RPL_ILK_BIT;
      A(;
      A     "DOOR_EXTRACTOR_DB".DOOR_EXT_MAN_SS;
      A(;
      O     "DOOR_EXTRACTOR_DB".MAIN_STK_UP_STA_PB;
      O     "DOOR_EXTRACTOR_DB".MAIN_STK_UP_CMD;
      );
      A     "DOOR_EXTRACTOR_DB".DOOR_EXT_STP_PB;
      O;
      A     "DOOR_EXTRACTOR_DB".DOOR_EXT_AUTO_SS;
      A     "DOOR_EXTRACTOR_DB".DR_EXT_AUTO_STA_BIT;
      A     "DOOR_EXTRACTOR_DB".DR_LCH_TURN_AUTO_DN_SET;
      A     "DOOR_EXTRACTOR_DB".DR_LCH_AUTO_DN_OVR;
      );
      A     "DOOR_EXTRACTOR_DB".SLEW_NR_FWD_OP_CUT;
      A     "DOOR_EXTRACTOR_DB".VER_COMP_FWD_OP_CUT;
      A     "DOOR_EXTRACTOR_DB".TRA_NOR_FWD_OP_CUT;
      A     "DOOR_EXTRACTOR_DB".PRE_STK_UP_OP_CUT;
      A     "DOOR_EXTRACTOR_DB".DR_SPNG_LK_OP_CUT;
      A     "DOOR_EXTRACTOR_DB".DR_LCH_DN_OP_CUT;
      O;
      A     "DOOR_EXTRACTOR_DB".DOOR_EXT_LOC_SS;
      A     "HYDRAULIC_FUNCTIONS_DB".HYD_SYS_RDY_BIT;
      A     "DOOR_EXTRACTOR_DB".MAIN_STK_UP_STA_PB_LCS;
      );
      AN    "DOOR_EXTRACTOR_DB".MAIN_STK_UP_OP_CUT;
      AN    "DOOR_EXTRACTOR_DB".MAIN_STK_DN_CMD;
      =     L 0.0;
      A     L 0.0;
      BLD   102;
      =     "DOOR_EXTRACTOR_DB".MAIN_STK_UP_CMD;
      A(;
      A     L 0.0;
      FN    "DOOR_EXTRACTOR_DB".PULSE_26;
      );
      A     "DOOR_EXTRACTOR_DB".DOOR_EXT_AUTO_SS;
      A     "DOOR_EXTRACTOR_DB".MAIN_STK_UP_OP_CUT;
      S     "DOOR_EXTRACTOR_DB".MAIN_STK_AUTO_FWD_SET;
      A     L 0.0;
      FP    "DOOR_EXTRACTOR_DB".PULSE_11;
      =     L 0.1;
      A     L 0.1;
      JNB   M047;
      L     0;
      T     "DOOR_EXTRACTOR_DB".MAIN_STK_UP_OP_CT_TM;
M047: NOP   0;
      A     L 0.1;
      JNB   M048;
      L     0;
      T     "DOOR_EXTRACTOR_DB".MAIN_STK_ATO_UP_DL_T;
M048: NOP   0;
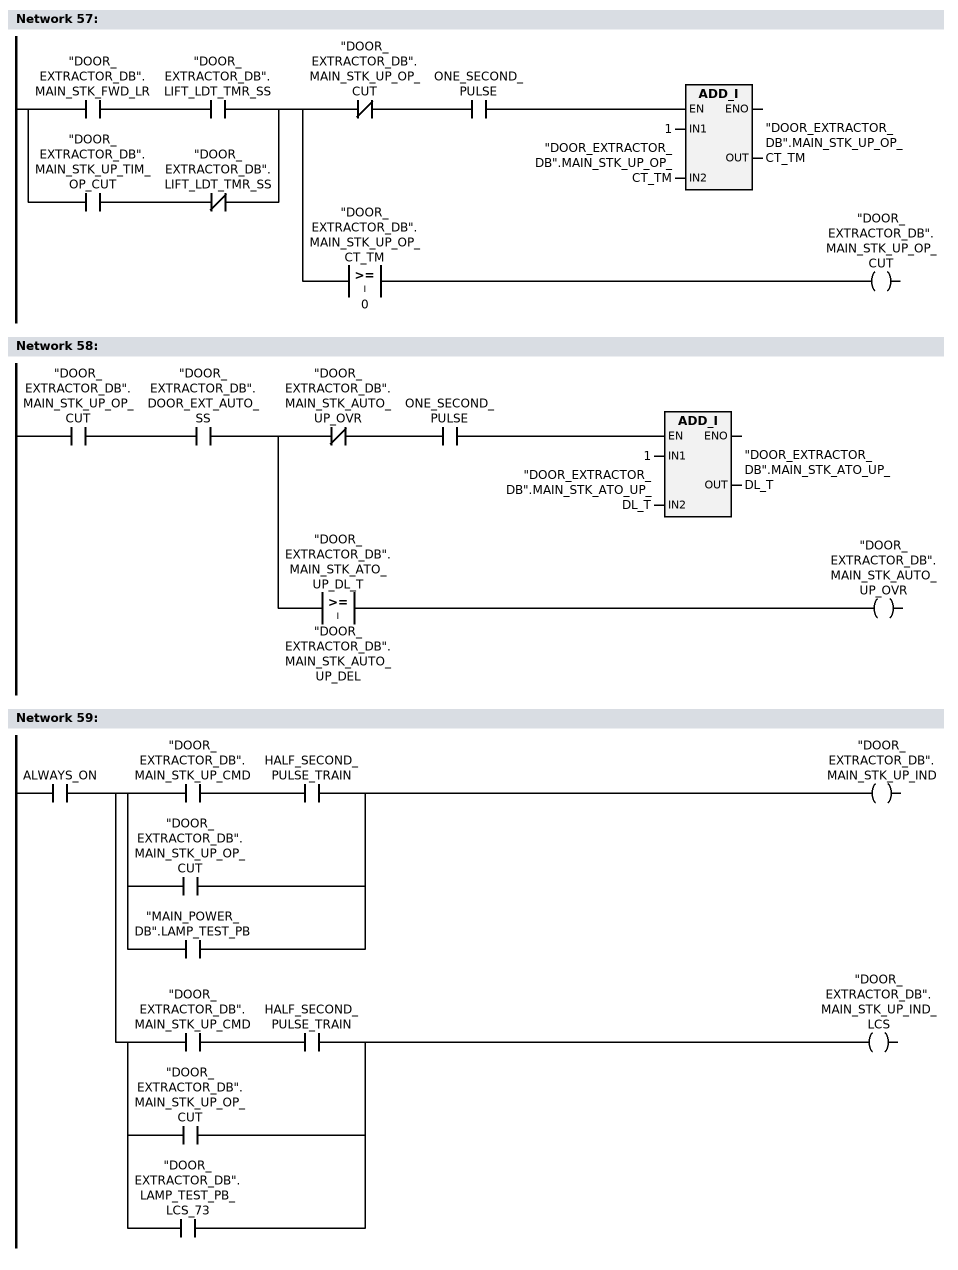
NETWORK
TITLE =
      A     "DOOR_EXTRACTOR_DB".MAIN_STK_FWD_LR;
      A     "DOOR_EXTRACTOR_DB".LIFT_LDT_TMR_SS;
      O;
      A     "DOOR_EXTRACTOR_DB".MAIN_STK_UP_TIM_OP_CUT;
      AN    "DOOR_EXTRACTOR_DB".LIFT_LDT_TMR_SS;
      =     L 0.0;
      A     L 0.0;
      AN    "DOOR_EXTRACTOR_DB".MAIN_STK_UP_OP_CUT;
      A     "ONE_SECOND_PULSE";
      JNB   M049;
      L     1;
      L     "DOOR_EXTRACTOR_DB".MAIN_STK_UP_OP_CT_TM;
      +I;
      T     "DOOR_EXTRACTOR_DB".MAIN_STK_UP_OP_CT_TM;
M049: NOP   0;
      A     L 0.0;
      A(;
      L     "DOOR_EXTRACTOR_DB".MAIN_STK_UP_OP_CT_TM;
      L     0;
      >=I;
      );
      =     "DOOR_EXTRACTOR_DB".MAIN_STK_UP_OP_CUT;
NETWORK
TITLE =
      A     "DOOR_EXTRACTOR_DB".MAIN_STK_UP_OP_CUT;
      A     "DOOR_EXTRACTOR_DB".DOOR_EXT_AUTO_SS;
      =     L 0.0;
      A     L 0.0;
      AN    "DOOR_EXTRACTOR_DB".MAIN_STK_AUTO_UP_OVR;
      A     "ONE_SECOND_PULSE";
      JNB   M050;
      L     1;
      L     "DOOR_EXTRACTOR_DB".MAIN_STK_ATO_UP_DL_T;
      +I;
      T     "DOOR_EXTRACTOR_DB".MAIN_STK_ATO_UP_DL_T;
M050: NOP   0;
      A     L 0.0;
      A(;
      L     "DOOR_EXTRACTOR_DB".MAIN_STK_ATO_UP_DL_T;
      L     "DOOR_EXTRACTOR_DB".MAIN_STK_AUTO_UP_DEL;
      >=I;
      );
      =     "DOOR_EXTRACTOR_DB".MAIN_STK_AUTO_UP_OVR;
NETWORK
TITLE =
      A     "ALWAYS_ON";
      =     L 0.0;
      A     L 0.0;
      A(;
      A     "DOOR_EXTRACTOR_DB".MAIN_STK_UP_CMD;
      A     "HALF_SECOND_PULSE_TRAIN";
      O     "DOOR_EXTRACTOR_DB".MAIN_STK_UP_OP_CUT;
      O     "MAIN_POWER_DB".LAMP_TEST_PB;
      );
      =     "DOOR_EXTRACTOR_DB".MAIN_STK_UP_IND;
      A     L 0.0;
      A(;
      A     "DOOR_EXTRACTOR_DB".MAIN_STK_UP_CMD;
      A     "HALF_SECOND_PULSE_TRAIN";
      O     "DOOR_EXTRACTOR_DB".MAIN_STK_UP_OP_CUT;
      O     "DOOR_EXTRACTOR_DB".LAMP_TEST_PB_LCS_73;
      );
      =     "DOOR_EXTRACTOR_DB".MAIN_STK_UP_IND_LCS;
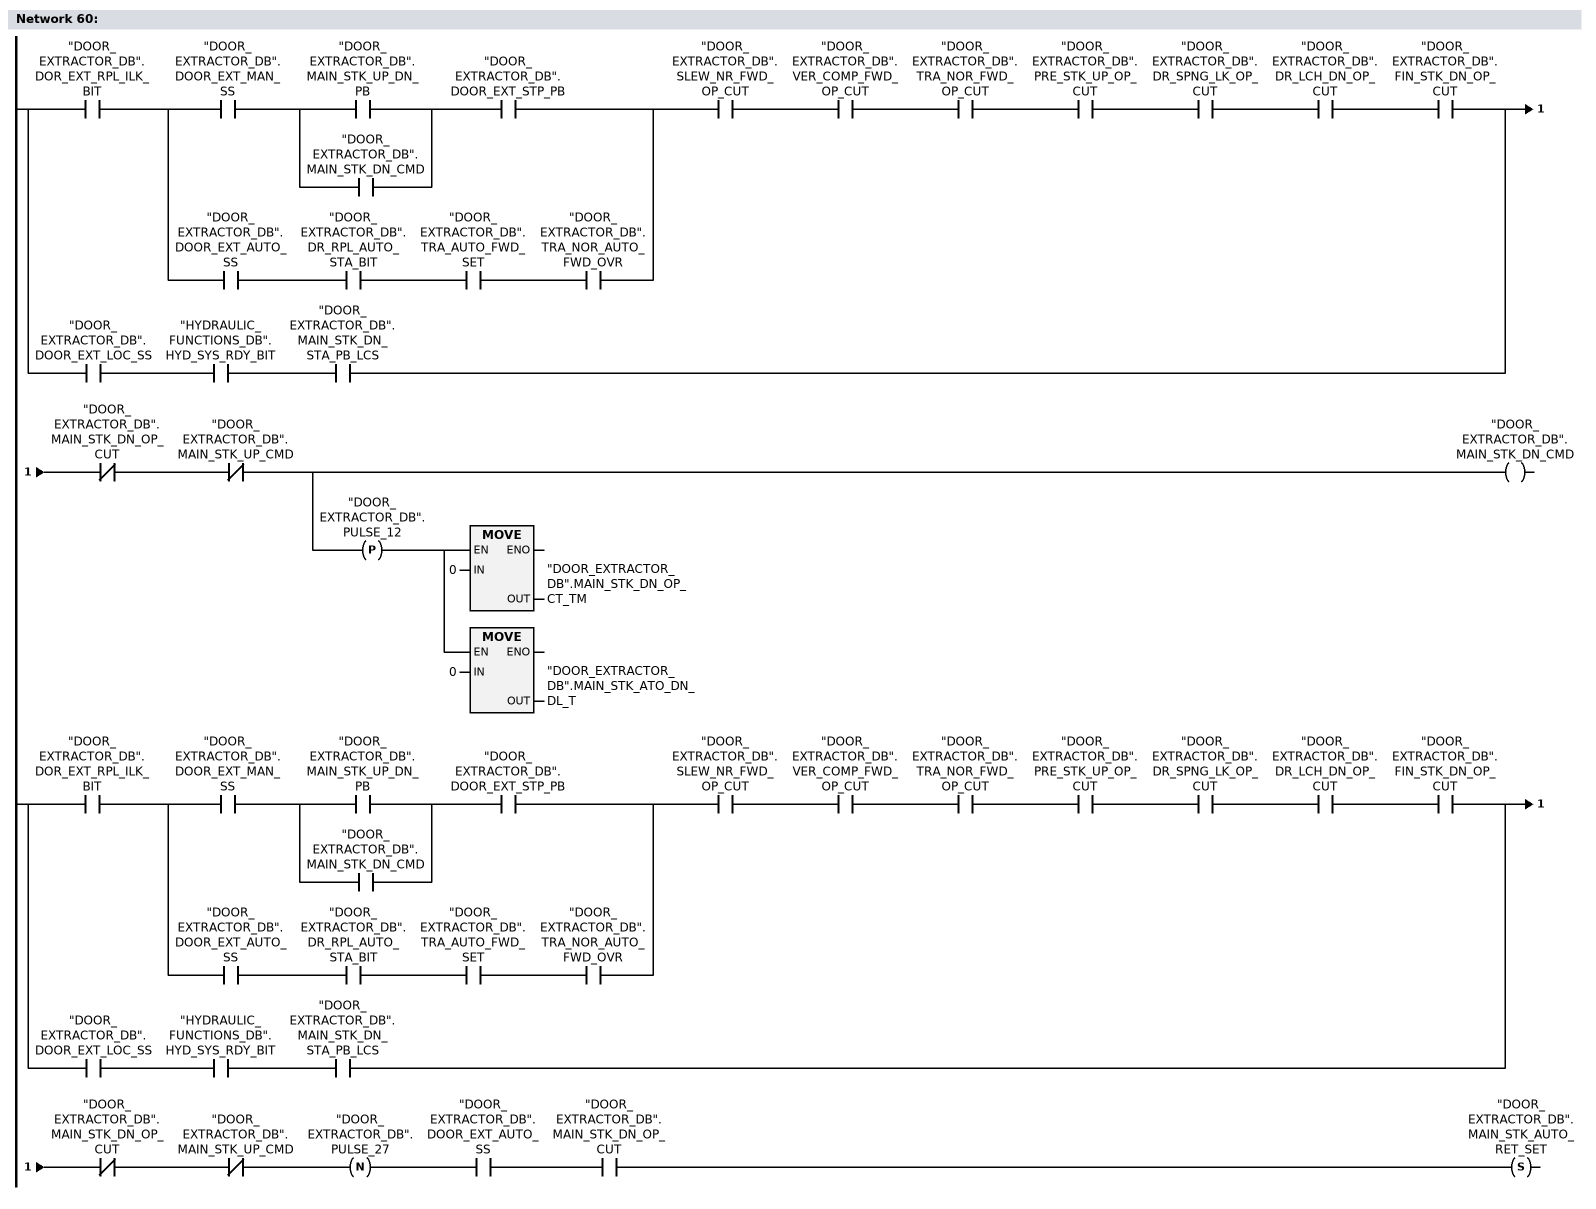
NETWORK
TITLE =
      A(;
      A     "DOOR_EXTRACTOR_DB".DOR_EXT_RPL_ILK_BIT;
      A(;
      A     "DOOR_EXTRACTOR_DB".DOOR_EXT_MAN_SS;
      A(;
      O     "DOOR_EXTRACTOR_DB".MAIN_STK_UP_DN_PB;
      O     "DOOR_EXTRACTOR_DB".MAIN_STK_DN_CMD;
      );
      A     "DOOR_EXTRACTOR_DB".DOOR_EXT_STP_PB;
      O;
      A     "DOOR_EXTRACTOR_DB".DOOR_EXT_AUTO_SS;
      A     "DOOR_EXTRACTOR_DB".DR_RPL_AUTO_STA_BIT;
      A     "DOOR_EXTRACTOR_DB".TRA_AUTO_FWD_SET;
      A     "DOOR_EXTRACTOR_DB".TRA_NOR_AUTO_FWD_OVR;
      );
      A     "DOOR_EXTRACTOR_DB".SLEW_NR_FWD_OP_CUT;
      A     "DOOR_EXTRACTOR_DB".VER_COMP_FWD_OP_CUT;
      A     "DOOR_EXTRACTOR_DB".TRA_NOR_FWD_OP_CUT;
      A     "DOOR_EXTRACTOR_DB".PRE_STK_UP_OP_CUT;
      A     "DOOR_EXTRACTOR_DB".DR_SPNG_LK_OP_CUT;
      A     "DOOR_EXTRACTOR_DB".DR_LCH_DN_OP_CUT;
      A     "DOOR_EXTRACTOR_DB".FIN_STK_DN_OP_CUT;
      O;
      A     "DOOR_EXTRACTOR_DB".DOOR_EXT_LOC_SS;
      A     "HYDRAULIC_FUNCTIONS_DB".HYD_SYS_RDY_BIT;
      A     "DOOR_EXTRACTOR_DB".MAIN_STK_DN_STA_PB_LCS;
      );
      AN    "DOOR_EXTRACTOR_DB".MAIN_STK_DN_OP_CUT;
      AN    "DOOR_EXTRACTOR_DB".MAIN_STK_UP_CMD;
      =     L 0.0;
      A     L 0.0;
      BLD   102;
      =     "DOOR_EXTRACTOR_DB".MAIN_STK_DN_CMD;
      A(;
      A     L 0.0;
      FN    "DOOR_EXTRACTOR_DB".PULSE_27;
      );
      A     "DOOR_EXTRACTOR_DB".DOOR_EXT_AUTO_SS;
      A     "DOOR_EXTRACTOR_DB".MAIN_STK_DN_OP_CUT;
      S     "DOOR_EXTRACTOR_DB".MAIN_STK_AUTO_RET_SET;
      A     L 0.0;
      FP    "DOOR_EXTRACTOR_DB".PULSE_12;
      =     L 0.1;
      A     L 0.1;
      JNB   M051;
      L     0;
      T     "DOOR_EXTRACTOR_DB".MAIN_STK_DN_OP_CT_TM;
M051: NOP   0;
      A     L 0.1;
      JNB   M052;
      L     0;
      T     "DOOR_EXTRACTOR_DB".MAIN_STK_ATO_DN_DL_T;
M052: NOP   0;
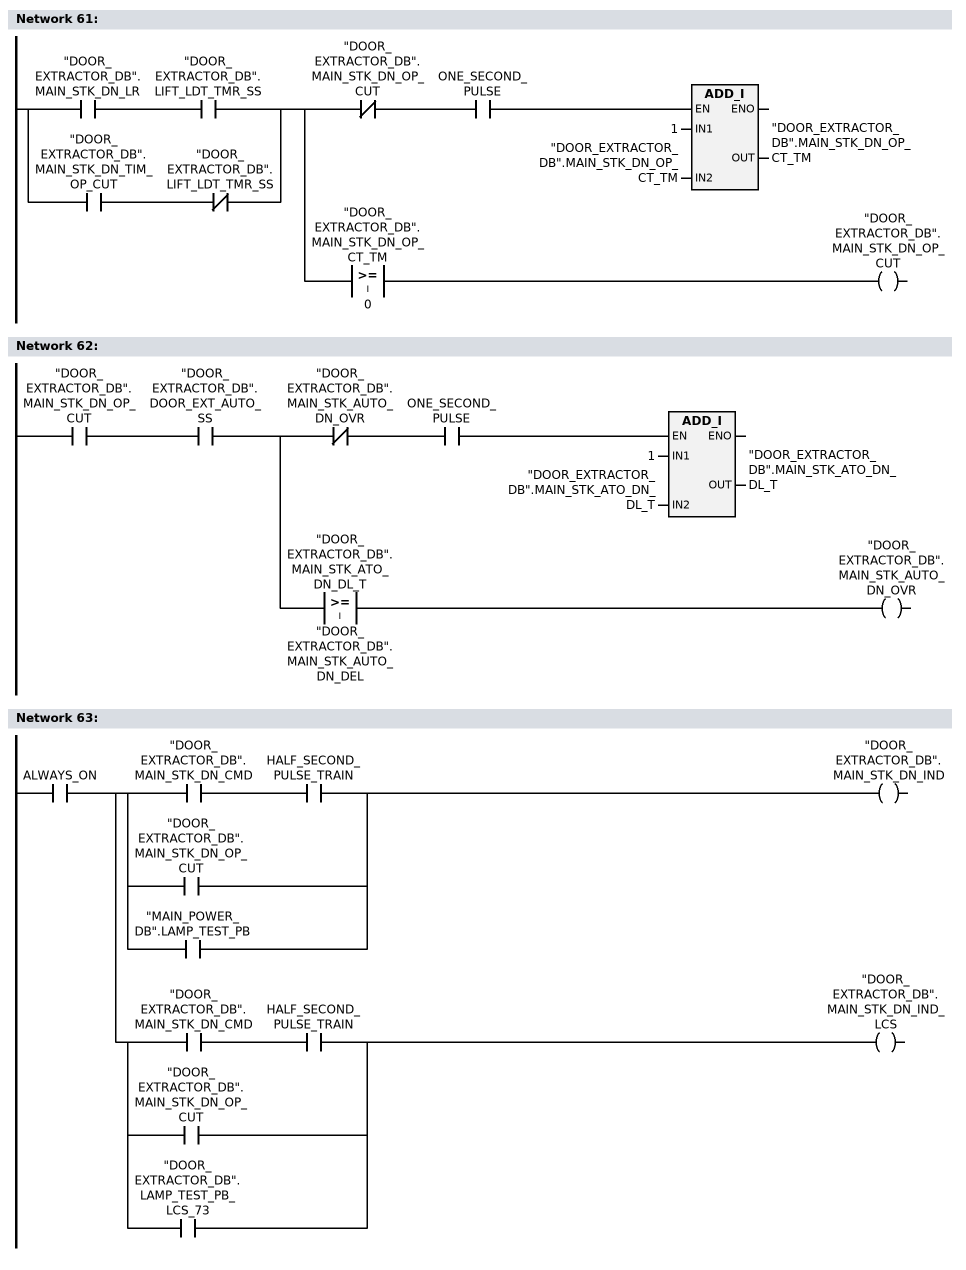
NETWORK
TITLE =
      A     "DOOR_EXTRACTOR_DB".MAIN_STK_DN_LR;
      A     "DOOR_EXTRACTOR_DB".LIFT_LDT_TMR_SS;
      O;
      A     "DOOR_EXTRACTOR_DB".MAIN_STK_DN_TIM_OP_CUT;
      AN    "DOOR_EXTRACTOR_DB".LIFT_LDT_TMR_SS;
      =     L 0.0;
      A     L 0.0;
      AN    "DOOR_EXTRACTOR_DB".MAIN_STK_DN_OP_CUT;
      A     "ONE_SECOND_PULSE";
      JNB   M053;
      L     1;
      L     "DOOR_EXTRACTOR_DB".MAIN_STK_DN_OP_CT_TM;
      +I;
      T     "DOOR_EXTRACTOR_DB".MAIN_STK_DN_OP_CT_TM;
M053: NOP   0;
      A     L 0.0;
      A(;
      L     "DOOR_EXTRACTOR_DB".MAIN_STK_DN_OP_CT_TM;
      L     0;
      >=I;
      );
      =     "DOOR_EXTRACTOR_DB".MAIN_STK_DN_OP_CUT;
NETWORK
TITLE =
      A     "DOOR_EXTRACTOR_DB".MAIN_STK_DN_OP_CUT;
      A     "DOOR_EXTRACTOR_DB".DOOR_EXT_AUTO_SS;
      =     L 0.0;
      A     L 0.0;
      AN    "DOOR_EXTRACTOR_DB".MAIN_STK_AUTO_DN_OVR;
      A     "ONE_SECOND_PULSE";
      JNB   M054;
      L     1;
      L     "DOOR_EXTRACTOR_DB".MAIN_STK_ATO_DN_DL_T;
      +I;
      T     "DOOR_EXTRACTOR_DB".MAIN_STK_ATO_DN_DL_T;
M054: NOP   0;
      A     L 0.0;
      A(;
      L     "DOOR_EXTRACTOR_DB".MAIN_STK_ATO_DN_DL_T;
      L     "DOOR_EXTRACTOR_DB".MAIN_STK_AUTO_DN_DEL;
      >=I;
      );
      =     "DOOR_EXTRACTOR_DB".MAIN_STK_AUTO_DN_OVR;
NETWORK
TITLE =
      A     "ALWAYS_ON";
      =     L 0.0;
      A     L 0.0;
      A(;
      A     "DOOR_EXTRACTOR_DB".MAIN_STK_DN_CMD;
      A     "HALF_SECOND_PULSE_TRAIN";
      O     "DOOR_EXTRACTOR_DB".MAIN_STK_DN_OP_CUT;
      O     "MAIN_POWER_DB".LAMP_TEST_PB;
      );
      =     "DOOR_EXTRACTOR_DB".MAIN_STK_DN_IND;
      A     L 0.0;
      A(;
      A     "DOOR_EXTRACTOR_DB".MAIN_STK_DN_CMD;
      A     "HALF_SECOND_PULSE_TRAIN";
      O     "DOOR_EXTRACTOR_DB".MAIN_STK_DN_OP_CUT;
      O     "DOOR_EXTRACTOR_DB".LAMP_TEST_PB_LCS_73;
      );
      =     "DOOR_EXTRACTOR_DB".MAIN_STK_DN_IND_LCS;
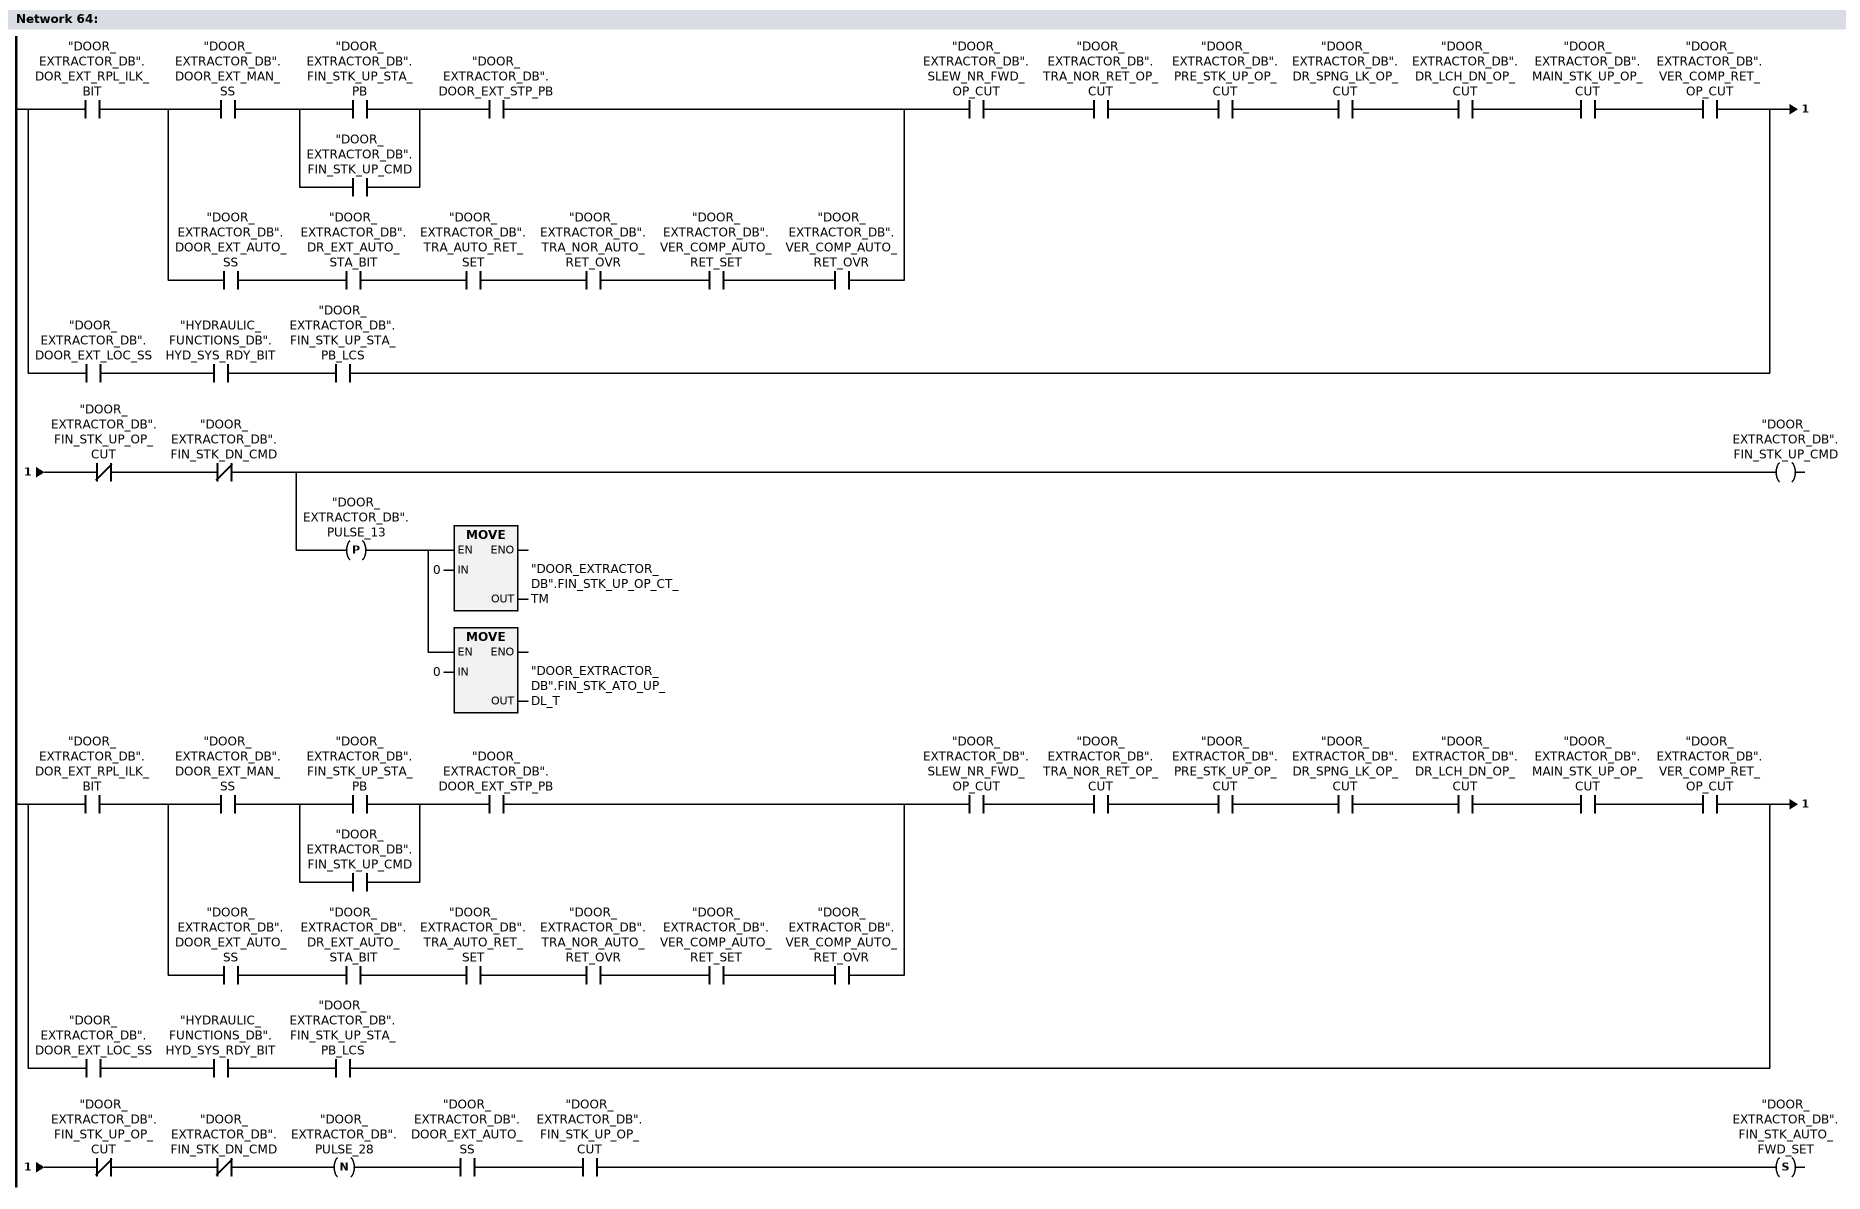
NETWORK
TITLE =
      A(;
      A     "DOOR_EXTRACTOR_DB".DOR_EXT_RPL_ILK_BIT;
      A(;
      A     "DOOR_EXTRACTOR_DB".DOOR_EXT_MAN_SS;
      A(;
      O     "DOOR_EXTRACTOR_DB".FIN_STK_UP_STA_PB;
      O     "DOOR_EXTRACTOR_DB".FIN_STK_UP_CMD;
      );
      A     "DOOR_EXTRACTOR_DB".DOOR_EXT_STP_PB;
      O;
      A     "DOOR_EXTRACTOR_DB".DOOR_EXT_AUTO_SS;
      A     "DOOR_EXTRACTOR_DB".DR_EXT_AUTO_STA_BIT;
      A     "DOOR_EXTRACTOR_DB".TRA_AUTO_RET_SET;
      A     "DOOR_EXTRACTOR_DB".TRA_NOR_AUTO_RET_OVR;
      A     "DOOR_EXTRACTOR_DB".VER_COMP_AUTO_RET_SET;
      A     "DOOR_EXTRACTOR_DB".VER_COMP_AUTO_RET_OVR;
      );
      A     "DOOR_EXTRACTOR_DB".SLEW_NR_FWD_OP_CUT;
      A     "DOOR_EXTRACTOR_DB".TRA_NOR_RET_OP_CUT;
      A     "DOOR_EXTRACTOR_DB".PRE_STK_UP_OP_CUT;
      A     "DOOR_EXTRACTOR_DB".DR_SPNG_LK_OP_CUT;
      A     "DOOR_EXTRACTOR_DB".DR_LCH_DN_OP_CUT;
      A     "DOOR_EXTRACTOR_DB".MAIN_STK_UP_OP_CUT;
      A     "DOOR_EXTRACTOR_DB".VER_COMP_RET_OP_CUT;
      O;
      A     "DOOR_EXTRACTOR_DB".DOOR_EXT_LOC_SS;
      A     "HYDRAULIC_FUNCTIONS_DB".HYD_SYS_RDY_BIT;
      A     "DOOR_EXTRACTOR_DB".FIN_STK_UP_STA_PB_LCS;
      );
      AN    "DOOR_EXTRACTOR_DB".FIN_STK_UP_OP_CUT;
      AN    "DOOR_EXTRACTOR_DB".FIN_STK_DN_CMD;
      =     L 0.0;
      A     L 0.0;
      BLD   102;
      =     "DOOR_EXTRACTOR_DB".FIN_STK_UP_CMD;
      A(;
      A     L 0.0;
      FN    "DOOR_EXTRACTOR_DB".PULSE_28;
      );
      A     "DOOR_EXTRACTOR_DB".DOOR_EXT_AUTO_SS;
      A     "DOOR_EXTRACTOR_DB".FIN_STK_UP_OP_CUT;
      S     "DOOR_EXTRACTOR_DB".FIN_STK_AUTO_FWD_SET;
      A     L 0.0;
      FP    "DOOR_EXTRACTOR_DB".PULSE_13;
      =     L 0.1;
      A     L 0.1;
      JNB   M055;
      L     0;
      T     "DOOR_EXTRACTOR_DB".FIN_STK_UP_OP_CT_TM;
M055: NOP   0;
      A     L 0.1;
      JNB   M056;
      L     0;
      T     "DOOR_EXTRACTOR_DB".FIN_STK_ATO_UP_DL_T;
M056: NOP   0;
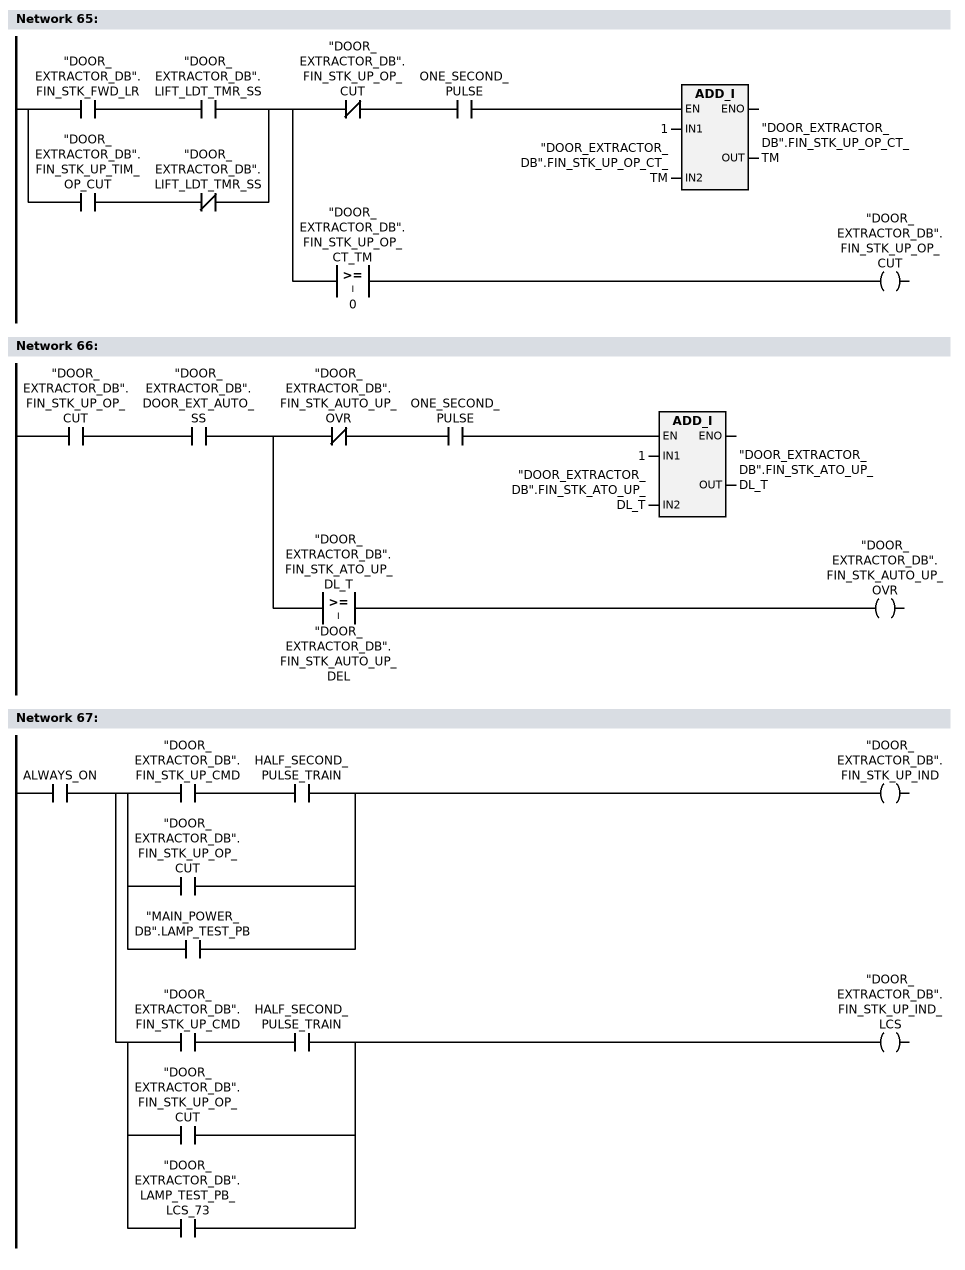
NETWORK
TITLE =
      A     "DOOR_EXTRACTOR_DB".FIN_STK_FWD_LR;
      A     "DOOR_EXTRACTOR_DB".LIFT_LDT_TMR_SS;
      O;
      A     "DOOR_EXTRACTOR_DB".FIN_STK_UP_TIM_OP_CUT;
      AN    "DOOR_EXTRACTOR_DB".LIFT_LDT_TMR_SS;
      =     L 0.0;
      A     L 0.0;
      AN    "DOOR_EXTRACTOR_DB".FIN_STK_UP_OP_CUT;
      A     "ONE_SECOND_PULSE";
      JNB   M057;
      L     1;
      L     "DOOR_EXTRACTOR_DB".FIN_STK_UP_OP_CT_TM;
      +I;
      T     "DOOR_EXTRACTOR_DB".FIN_STK_UP_OP_CT_TM;
M057: NOP   0;
      A     L 0.0;
      A(;
      L     "DOOR_EXTRACTOR_DB".FIN_STK_UP_OP_CT_TM;
      L     0;
      >=I;
      );
      =     "DOOR_EXTRACTOR_DB".FIN_STK_UP_OP_CUT;
NETWORK
TITLE =
      A     "DOOR_EXTRACTOR_DB".FIN_STK_UP_OP_CUT;
      A     "DOOR_EXTRACTOR_DB".DOOR_EXT_AUTO_SS;
      =     L 0.0;
      A     L 0.0;
      AN    "DOOR_EXTRACTOR_DB".FIN_STK_AUTO_UP_OVR;
      A     "ONE_SECOND_PULSE";
      JNB   M058;
      L     1;
      L     "DOOR_EXTRACTOR_DB".FIN_STK_ATO_UP_DL_T;
      +I;
      T     "DOOR_EXTRACTOR_DB".FIN_STK_ATO_UP_DL_T;
M058: NOP   0;
      A     L 0.0;
      A(;
      L     "DOOR_EXTRACTOR_DB".FIN_STK_ATO_UP_DL_T;
      L     "DOOR_EXTRACTOR_DB".FIN_STK_AUTO_UP_DEL;
      >=I;
      );
      =     "DOOR_EXTRACTOR_DB".FIN_STK_AUTO_UP_OVR;
NETWORK
TITLE =
      A     "ALWAYS_ON";
      =     L 0.0;
      A     L 0.0;
      A(;
      A     "DOOR_EXTRACTOR_DB".FIN_STK_UP_CMD;
      A     "HALF_SECOND_PULSE_TRAIN";
      O     "DOOR_EXTRACTOR_DB".FIN_STK_UP_OP_CUT;
      O     "MAIN_POWER_DB".LAMP_TEST_PB;
      );
      =     "DOOR_EXTRACTOR_DB".FIN_STK_UP_IND;
      A     L 0.0;
      A(;
      A     "DOOR_EXTRACTOR_DB".FIN_STK_UP_CMD;
      A     "HALF_SECOND_PULSE_TRAIN";
      O     "DOOR_EXTRACTOR_DB".FIN_STK_UP_OP_CUT;
      O     "DOOR_EXTRACTOR_DB".LAMP_TEST_PB_LCS_73;
      );
      =     "DOOR_EXTRACTOR_DB".FIN_STK_UP_IND_LCS;
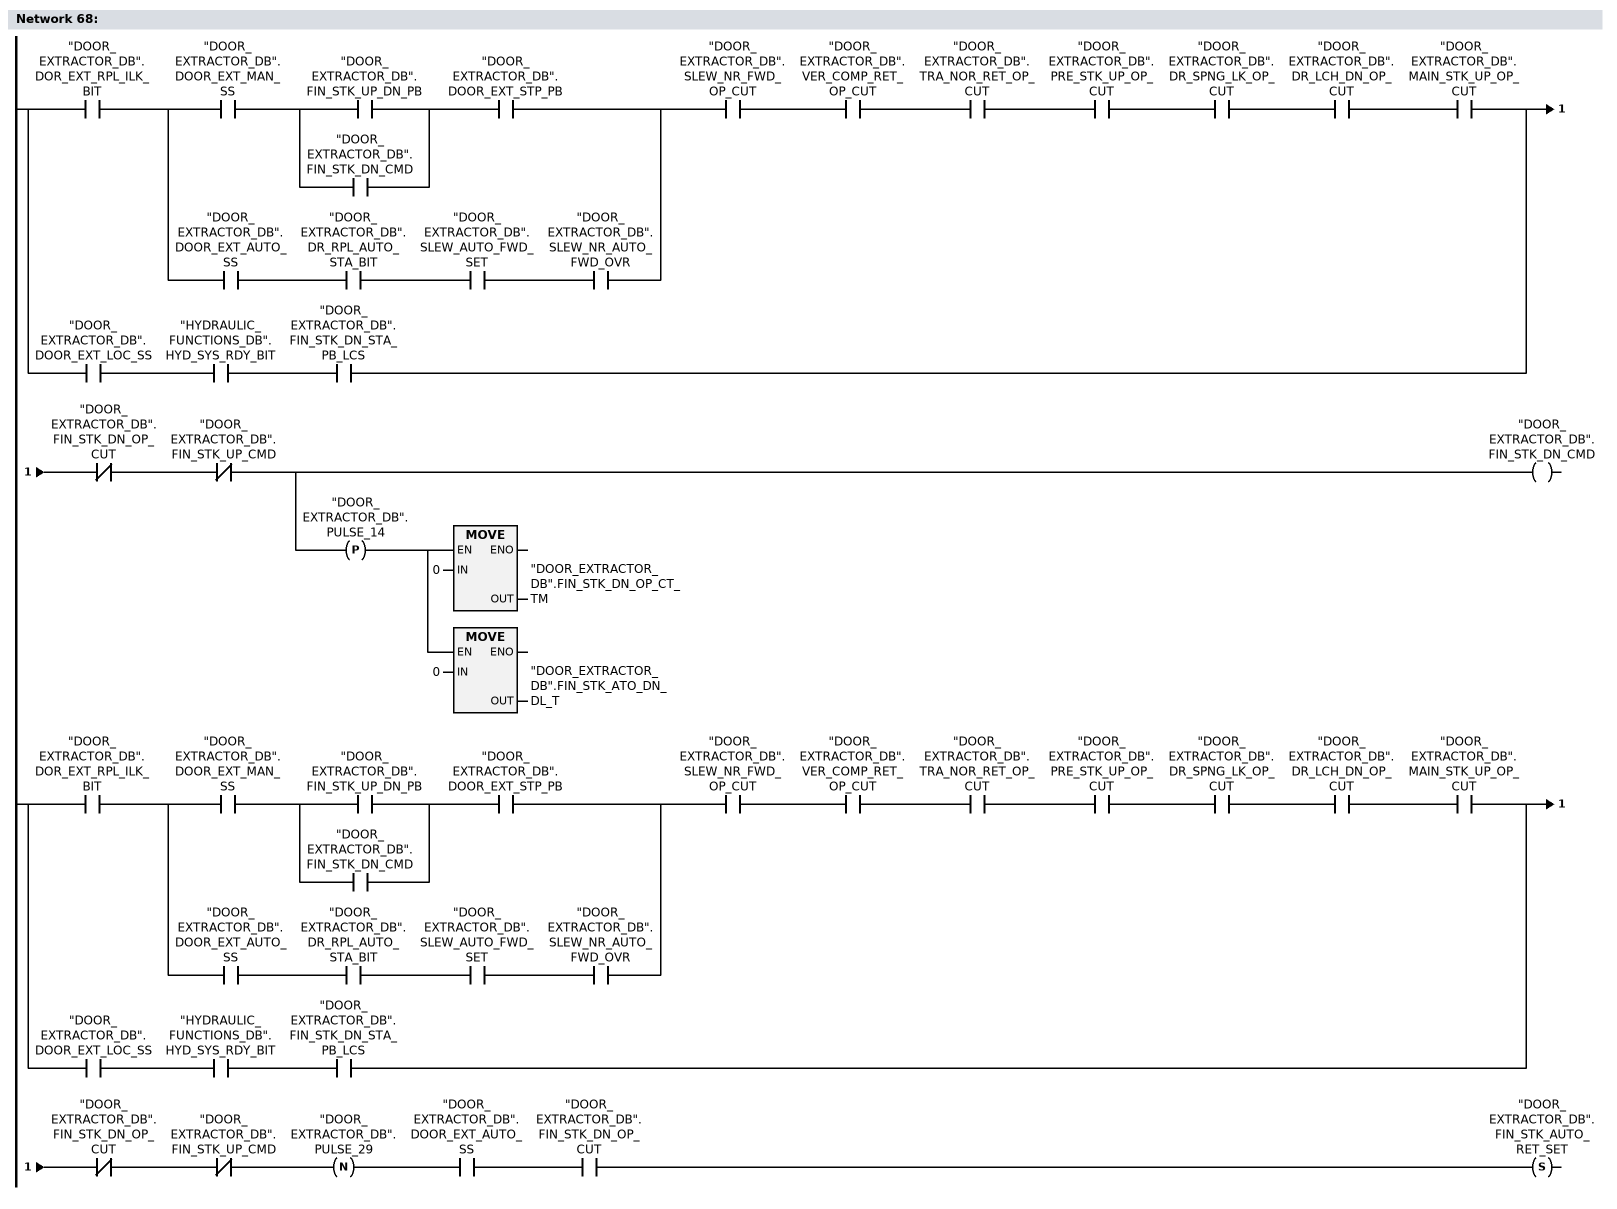
NETWORK
TITLE =
      A(;
      A     "DOOR_EXTRACTOR_DB".DOR_EXT_RPL_ILK_BIT;
      A(;
      A     "DOOR_EXTRACTOR_DB".DOOR_EXT_MAN_SS;
      A(;
      O     "DOOR_EXTRACTOR_DB".FIN_STK_UP_DN_PB;
      O     "DOOR_EXTRACTOR_DB".FIN_STK_DN_CMD;
      );
      A     "DOOR_EXTRACTOR_DB".DOOR_EXT_STP_PB;
      O;
      A     "DOOR_EXTRACTOR_DB".DOOR_EXT_AUTO_SS;
      A     "DOOR_EXTRACTOR_DB".DR_RPL_AUTO_STA_BIT;
      A     "DOOR_EXTRACTOR_DB".SLEW_AUTO_FWD_SET;
      A     "DOOR_EXTRACTOR_DB".SLEW_NR_AUTO_FWD_OVR;
      );
      A     "DOOR_EXTRACTOR_DB".SLEW_NR_FWD_OP_CUT;
      A     "DOOR_EXTRACTOR_DB".VER_COMP_RET_OP_CUT;
      A     "DOOR_EXTRACTOR_DB".TRA_NOR_RET_OP_CUT;
      A     "DOOR_EXTRACTOR_DB".PRE_STK_UP_OP_CUT;
      A     "DOOR_EXTRACTOR_DB".DR_SPNG_LK_OP_CUT;
      A     "DOOR_EXTRACTOR_DB".DR_LCH_DN_OP_CUT;
      A     "DOOR_EXTRACTOR_DB".MAIN_STK_UP_OP_CUT;
      O;
      A     "DOOR_EXTRACTOR_DB".DOOR_EXT_LOC_SS;
      A     "HYDRAULIC_FUNCTIONS_DB".HYD_SYS_RDY_BIT;
      A     "DOOR_EXTRACTOR_DB".FIN_STK_DN_STA_PB_LCS;
      );
      AN    "DOOR_EXTRACTOR_DB".FIN_STK_DN_OP_CUT;
      AN    "DOOR_EXTRACTOR_DB".FIN_STK_UP_CMD;
      =     L 0.0;
      A     L 0.0;
      BLD   102;
      =     "DOOR_EXTRACTOR_DB".FIN_STK_DN_CMD;
      A(;
      A     L 0.0;
      FN    "DOOR_EXTRACTOR_DB".PULSE_29;
      );
      A     "DOOR_EXTRACTOR_DB".DOOR_EXT_AUTO_SS;
      A     "DOOR_EXTRACTOR_DB".FIN_STK_DN_OP_CUT;
      S     "DOOR_EXTRACTOR_DB".FIN_STK_AUTO_RET_SET;
      A     L 0.0;
      FP    "DOOR_EXTRACTOR_DB".PULSE_14;
      =     L 0.1;
      A     L 0.1;
      JNB   M059;
      L     0;
      T     "DOOR_EXTRACTOR_DB".FIN_STK_DN_OP_CT_TM;
M059: NOP   0;
      A     L 0.1;
      JNB   M060;
      L     0;
      T     "DOOR_EXTRACTOR_DB".FIN_STK_ATO_DN_DL_T;
M060: NOP   0;
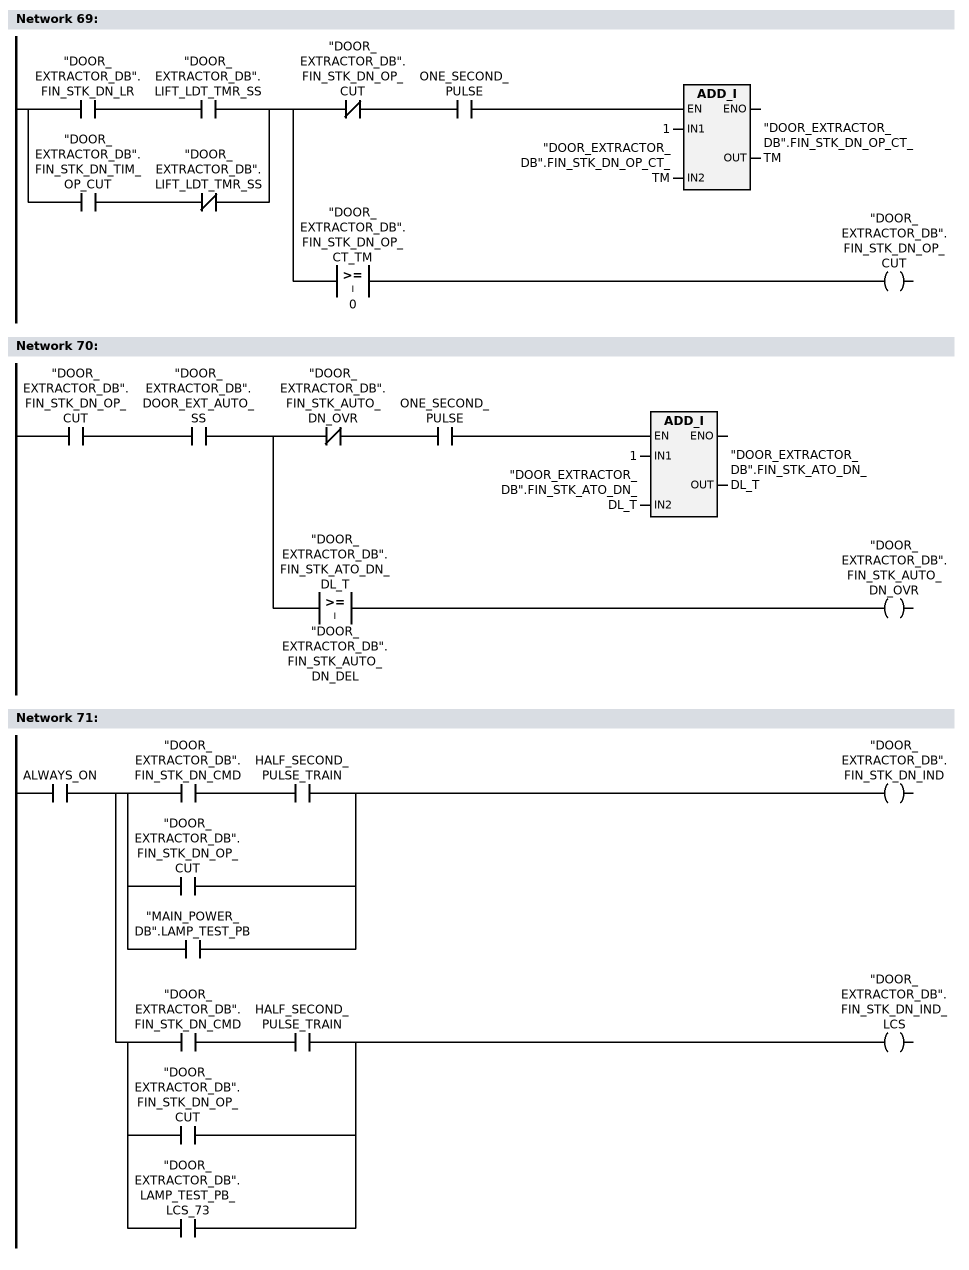
NETWORK
TITLE =
      A     "DOOR_EXTRACTOR_DB".FIN_STK_DN_LR;
      A     "DOOR_EXTRACTOR_DB".LIFT_LDT_TMR_SS;
      O;
      A     "DOOR_EXTRACTOR_DB".FIN_STK_DN_TIM_OP_CUT;
      AN    "DOOR_EXTRACTOR_DB".LIFT_LDT_TMR_SS;
      =     L 0.0;
      A     L 0.0;
      AN    "DOOR_EXTRACTOR_DB".FIN_STK_DN_OP_CUT;
      A     "ONE_SECOND_PULSE";
      JNB   M061;
      L     1;
      L     "DOOR_EXTRACTOR_DB".FIN_STK_DN_OP_CT_TM;
      +I;
      T     "DOOR_EXTRACTOR_DB".FIN_STK_DN_OP_CT_TM;
M061: NOP   0;
      A     L 0.0;
      A(;
      L     "DOOR_EXTRACTOR_DB".FIN_STK_DN_OP_CT_TM;
      L     0;
      >=I;
      );
      =     "DOOR_EXTRACTOR_DB".FIN_STK_DN_OP_CUT;
NETWORK
TITLE =
      A     "DOOR_EXTRACTOR_DB".FIN_STK_DN_OP_CUT;
      A     "DOOR_EXTRACTOR_DB".DOOR_EXT_AUTO_SS;
      =     L 0.0;
      A     L 0.0;
      AN    "DOOR_EXTRACTOR_DB".FIN_STK_AUTO_DN_OVR;
      A     "ONE_SECOND_PULSE";
      JNB   M062;
      L     1;
      L     "DOOR_EXTRACTOR_DB".FIN_STK_ATO_DN_DL_T;
      +I;
      T     "DOOR_EXTRACTOR_DB".FIN_STK_ATO_DN_DL_T;
M062: NOP   0;
      A     L 0.0;
      A(;
      L     "DOOR_EXTRACTOR_DB".FIN_STK_ATO_DN_DL_T;
      L     "DOOR_EXTRACTOR_DB".FIN_STK_AUTO_DN_DEL;
      >=I;
      );
      =     "DOOR_EXTRACTOR_DB".FIN_STK_AUTO_DN_OVR;
NETWORK
TITLE =
      A     "ALWAYS_ON";
      =     L 0.0;
      A     L 0.0;
      A(;
      A     "DOOR_EXTRACTOR_DB".FIN_STK_DN_CMD;
      A     "HALF_SECOND_PULSE_TRAIN";
      O     "DOOR_EXTRACTOR_DB".FIN_STK_DN_OP_CUT;
      O     "MAIN_POWER_DB".LAMP_TEST_PB;
      );
      =     "DOOR_EXTRACTOR_DB".FIN_STK_DN_IND;
      A     L 0.0;
      A(;
      A     "DOOR_EXTRACTOR_DB".FIN_STK_DN_CMD;
      A     "HALF_SECOND_PULSE_TRAIN";
      O     "DOOR_EXTRACTOR_DB".FIN_STK_DN_OP_CUT;
      O     "DOOR_EXTRACTOR_DB".LAMP_TEST_PB_LCS_73;
      );
      =     "DOOR_EXTRACTOR_DB".FIN_STK_DN_IND_LCS;
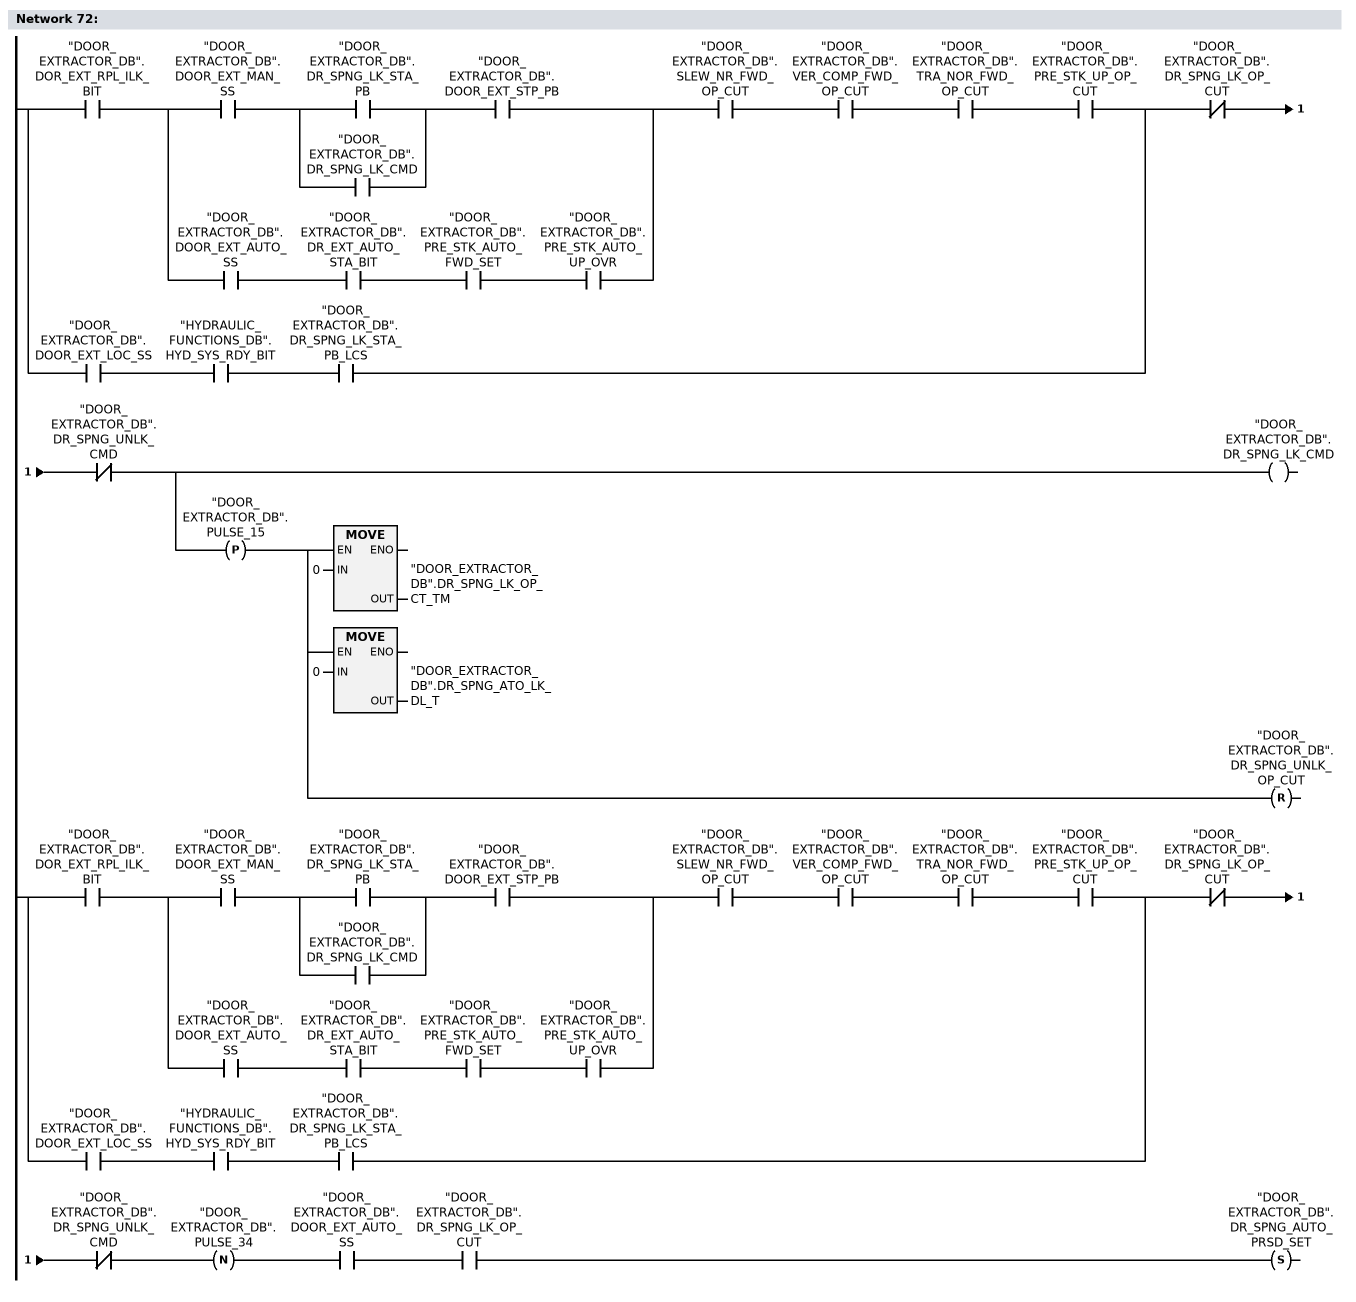
NETWORK
TITLE =
      A(;
      A     "DOOR_EXTRACTOR_DB".DOR_EXT_RPL_ILK_BIT;
      A(;
      A     "DOOR_EXTRACTOR_DB".DOOR_EXT_MAN_SS;
      A(;
      O     "DOOR_EXTRACTOR_DB".DR_SPNG_LK_STA_PB;
      O     "DOOR_EXTRACTOR_DB".DR_SPNG_LK_CMD;
      );
      A     "DOOR_EXTRACTOR_DB".DOOR_EXT_STP_PB;
      O;
      A     "DOOR_EXTRACTOR_DB".DOOR_EXT_AUTO_SS;
      A     "DOOR_EXTRACTOR_DB".DR_EXT_AUTO_STA_BIT;
      A     "DOOR_EXTRACTOR_DB".PRE_STK_AUTO_FWD_SET;
      A     "DOOR_EXTRACTOR_DB".PRE_STK_AUTO_UP_OVR;
      );
      A     "DOOR_EXTRACTOR_DB".SLEW_NR_FWD_OP_CUT;
      A     "DOOR_EXTRACTOR_DB".VER_COMP_FWD_OP_CUT;
      A     "DOOR_EXTRACTOR_DB".TRA_NOR_FWD_OP_CUT;
      A     "DOOR_EXTRACTOR_DB".PRE_STK_UP_OP_CUT;
      O;
      A     "DOOR_EXTRACTOR_DB".DOOR_EXT_LOC_SS;
      A     "HYDRAULIC_FUNCTIONS_DB".HYD_SYS_RDY_BIT;
      A     "DOOR_EXTRACTOR_DB".DR_SPNG_LK_STA_PB_LCS;
      );
      AN    "DOOR_EXTRACTOR_DB".DR_SPNG_LK_OP_CUT;
      AN    "DOOR_EXTRACTOR_DB".DR_SPNG_UNLK_CMD;
      =     L 0.0;
      A     L 0.0;
      BLD   102;
      =     "DOOR_EXTRACTOR_DB".DR_SPNG_LK_CMD;
      A(;
      A     L 0.0;
      FN    "DOOR_EXTRACTOR_DB".PULSE_34;
      );
      A     "DOOR_EXTRACTOR_DB".DOOR_EXT_AUTO_SS;
      A     "DOOR_EXTRACTOR_DB".DR_SPNG_LK_OP_CUT;
      S     "DOOR_EXTRACTOR_DB".DR_SPNG_AUTO_PRSD_SET;
      A     L 0.0;
      FP    "DOOR_EXTRACTOR_DB".PULSE_15;
      =     L 0.1;
      A     L 0.1;
      JNB   M063;
      L     0;
      T     "DOOR_EXTRACTOR_DB".DR_SPNG_LK_OP_CT_TM;
M063: NOP   0;
      A     L 0.1;
      JNB   M064;
      L     0;
      T     "DOOR_EXTRACTOR_DB".DR_SPNG_ATO_LK_DL_T;
M064: NOP   0;
      A     L 0.1;
      BLD   102;
      R     "DOOR_EXTRACTOR_DB".DR_SPNG_UNLK_OP_CUT;
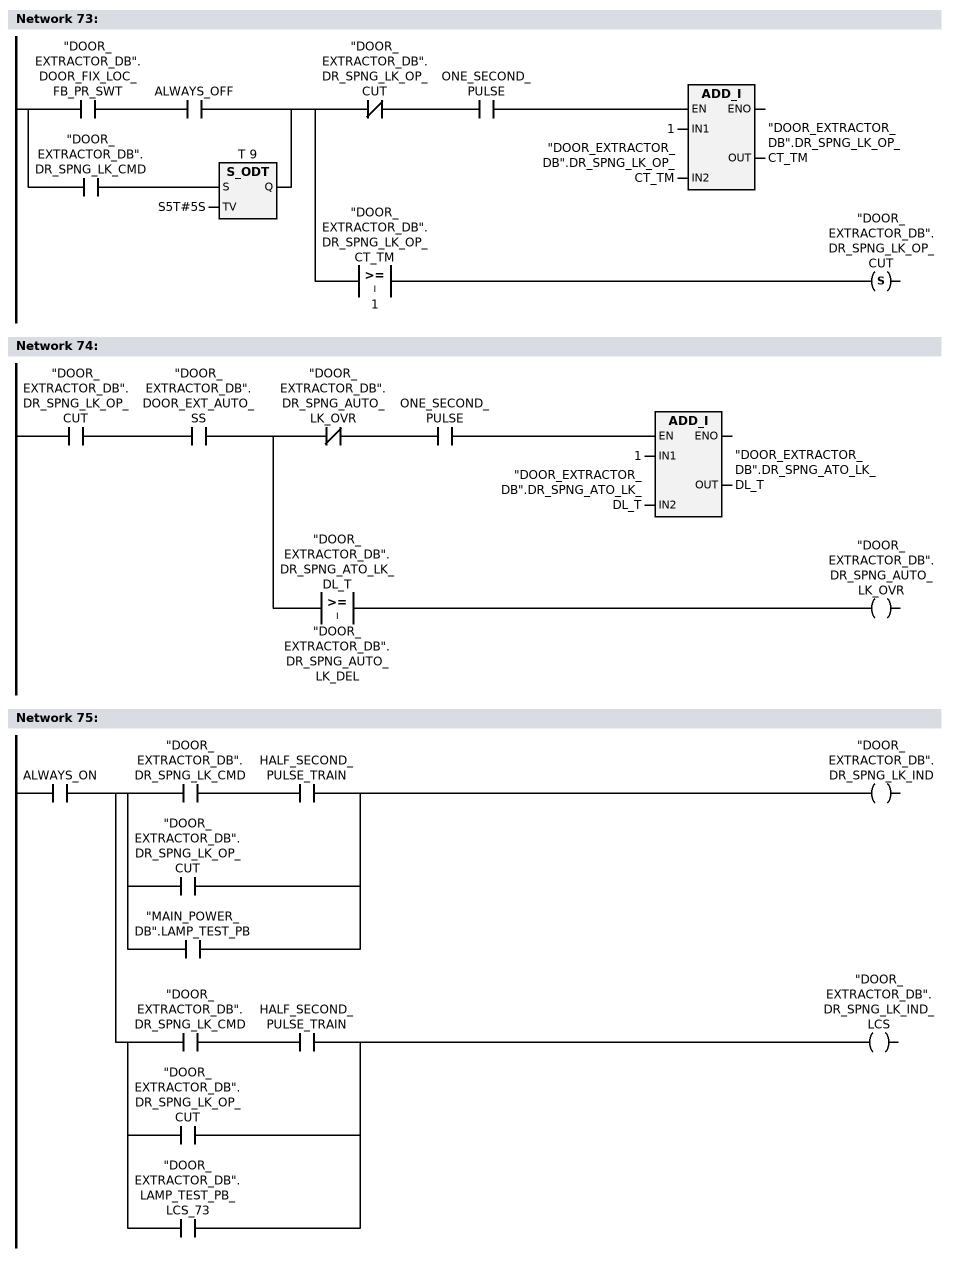
NETWORK
TITLE =
      A     "DOOR_EXTRACTOR_DB".DOOR_FIX_LOC_FB_PR_SWT;
      A     "ALWAYS_OFF";
      O(;
      A     "DOOR_EXTRACTOR_DB".DR_SPNG_LK_CMD;
      L     S5T#5S;
      SD    T 9;
      NOP   0;
      NOP   0;
      NOP   0;
      A     T 9;
      );
      =     L 0.0;
      A     L 0.0;
      AN    "DOOR_EXTRACTOR_DB".DR_SPNG_LK_OP_CUT;
      A     "ONE_SECOND_PULSE";
      JNB   M065;
      L     1;
      L     "DOOR_EXTRACTOR_DB".DR_SPNG_LK_OP_CT_TM;
      +I;
      T     "DOOR_EXTRACTOR_DB".DR_SPNG_LK_OP_CT_TM;
M065: NOP   0;
      A     L 0.0;
      A(;
      L     "DOOR_EXTRACTOR_DB".DR_SPNG_LK_OP_CT_TM;
      L     1;
      >=I;
      );
      S     "DOOR_EXTRACTOR_DB".DR_SPNG_LK_OP_CUT;
NETWORK
TITLE =
      A     "DOOR_EXTRACTOR_DB".DR_SPNG_LK_OP_CUT;
      A     "DOOR_EXTRACTOR_DB".DOOR_EXT_AUTO_SS;
      =     L 0.0;
      A     L 0.0;
      AN    "DOOR_EXTRACTOR_DB".DR_SPNG_AUTO_LK_OVR;
      A     "ONE_SECOND_PULSE";
      JNB   M066;
      L     1;
      L     "DOOR_EXTRACTOR_DB".DR_SPNG_ATO_LK_DL_T;
      +I;
      T     "DOOR_EXTRACTOR_DB".DR_SPNG_ATO_LK_DL_T;
M066: NOP   0;
      A     L 0.0;
      A(;
      L     "DOOR_EXTRACTOR_DB".DR_SPNG_ATO_LK_DL_T;
      L     "DOOR_EXTRACTOR_DB".DR_SPNG_AUTO_LK_DEL;
      >=I;
      );
      =     "DOOR_EXTRACTOR_DB".DR_SPNG_AUTO_LK_OVR;
NETWORK
TITLE =
      A     "ALWAYS_ON";
      =     L 0.0;
      A     L 0.0;
      A(;
      A     "DOOR_EXTRACTOR_DB".DR_SPNG_LK_CMD;
      A     "HALF_SECOND_PULSE_TRAIN";
      O     "DOOR_EXTRACTOR_DB".DR_SPNG_LK_OP_CUT;
      O     "MAIN_POWER_DB".LAMP_TEST_PB;
      );
      =     "DOOR_EXTRACTOR_DB".DR_SPNG_LK_IND;
      A     L 0.0;
      A(;
      A     "DOOR_EXTRACTOR_DB".DR_SPNG_LK_CMD;
      A     "HALF_SECOND_PULSE_TRAIN";
      O     "DOOR_EXTRACTOR_DB".DR_SPNG_LK_OP_CUT;
      O     "DOOR_EXTRACTOR_DB".LAMP_TEST_PB_LCS_73;
      );
      =     "DOOR_EXTRACTOR_DB".DR_SPNG_LK_IND_LCS;
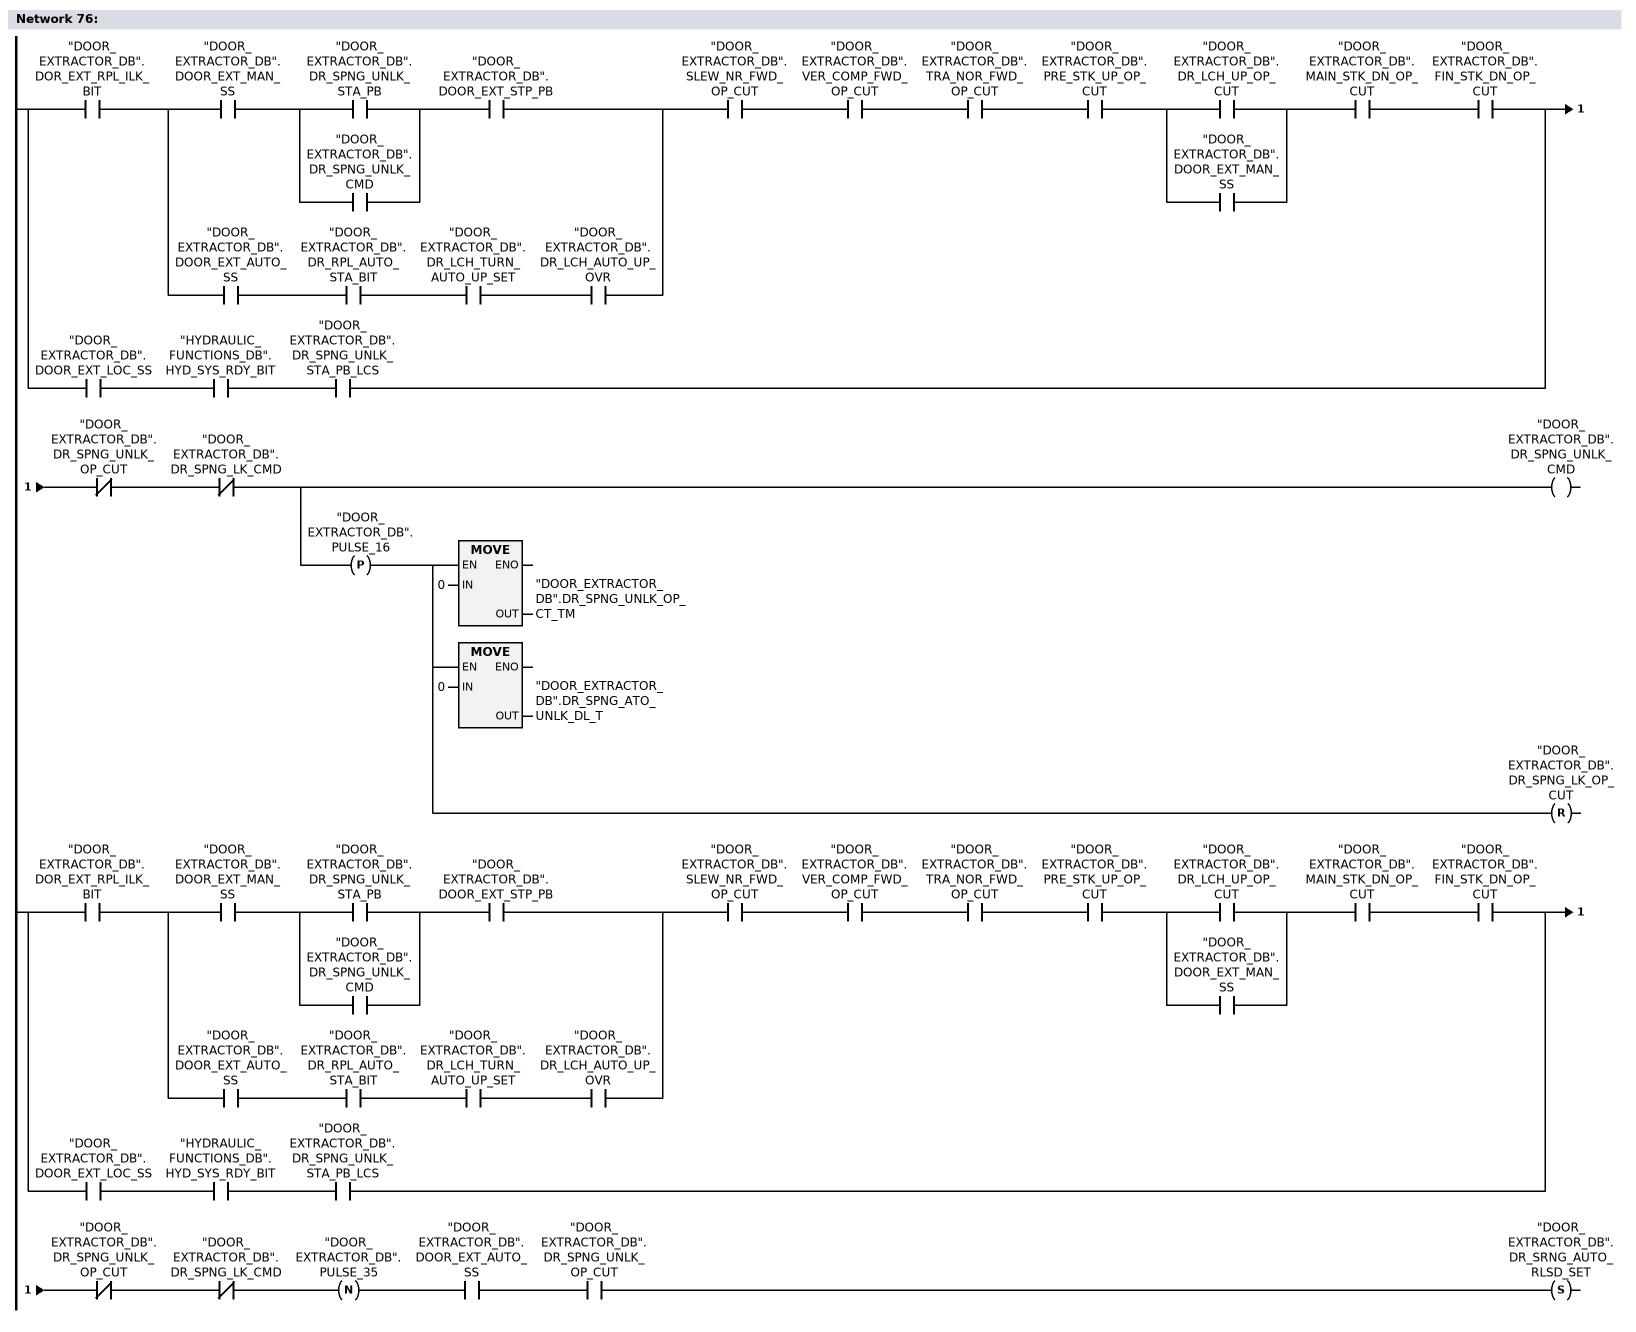
NETWORK
TITLE =
      A(;
      A     "DOOR_EXTRACTOR_DB".DOR_EXT_RPL_ILK_BIT;
      A(;
      A     "DOOR_EXTRACTOR_DB".DOOR_EXT_MAN_SS;
      A(;
      O     "DOOR_EXTRACTOR_DB".DR_SPNG_UNLK_STA_PB;
      O     "DOOR_EXTRACTOR_DB".DR_SPNG_UNLK_CMD;
      );
      A     "DOOR_EXTRACTOR_DB".DOOR_EXT_STP_PB;
      O;
      A     "DOOR_EXTRACTOR_DB".DOOR_EXT_AUTO_SS;
      A     "DOOR_EXTRACTOR_DB".DR_RPL_AUTO_STA_BIT;
      A     "DOOR_EXTRACTOR_DB".DR_LCH_TURN_AUTO_UP_SET;
      A     "DOOR_EXTRACTOR_DB".DR_LCH_AUTO_UP_OVR;
      );
      A     "DOOR_EXTRACTOR_DB".SLEW_NR_FWD_OP_CUT;
      A     "DOOR_EXTRACTOR_DB".VER_COMP_FWD_OP_CUT;
      A     "DOOR_EXTRACTOR_DB".TRA_NOR_FWD_OP_CUT;
      A     "DOOR_EXTRACTOR_DB".PRE_STK_UP_OP_CUT;
      A(;
      O     "DOOR_EXTRACTOR_DB".DR_LCH_UP_OP_CUT;
      O     "DOOR_EXTRACTOR_DB".DOOR_EXT_MAN_SS;
      );
      A     "DOOR_EXTRACTOR_DB".MAIN_STK_DN_OP_CUT;
      A     "DOOR_EXTRACTOR_DB".FIN_STK_DN_OP_CUT;
      O;
      A     "DOOR_EXTRACTOR_DB".DOOR_EXT_LOC_SS;
      A     "HYDRAULIC_FUNCTIONS_DB".HYD_SYS_RDY_BIT;
      A     "DOOR_EXTRACTOR_DB".DR_SPNG_UNLK_STA_PB_LCS;
      );
      AN    "DOOR_EXTRACTOR_DB".DR_SPNG_UNLK_OP_CUT;
      AN    "DOOR_EXTRACTOR_DB".DR_SPNG_LK_CMD;
      =     L 0.0;
      A     L 0.0;
      BLD   102;
      =     "DOOR_EXTRACTOR_DB".DR_SPNG_UNLK_CMD;
      A(;
      A     L 0.0;
      FN    "DOOR_EXTRACTOR_DB".PULSE_35;
      );
      A     "DOOR_EXTRACTOR_DB".DOOR_EXT_AUTO_SS;
      A     "DOOR_EXTRACTOR_DB".DR_SPNG_UNLK_OP_CUT;
      S     "DOOR_EXTRACTOR_DB".DR_SRNG_AUTO_RLSD_SET;
      A     L 0.0;
      FP    "DOOR_EXTRACTOR_DB".PULSE_16;
      =     L 0.1;
      A     L 0.1;
      JNB   M067;
      L     0;
      T     "DOOR_EXTRACTOR_DB".DR_SPNG_UNLK_OP_CT_TM;
M067: NOP   0;
      A     L 0.1;
      JNB   M068;
      L     0;
      T     "DOOR_EXTRACTOR_DB".DR_SPNG_ATO_UNLK_DL_T;
M068: NOP   0;
      A     L 0.1;
      BLD   102;
      R     "DOOR_EXTRACTOR_DB".DR_SPNG_LK_OP_CUT;
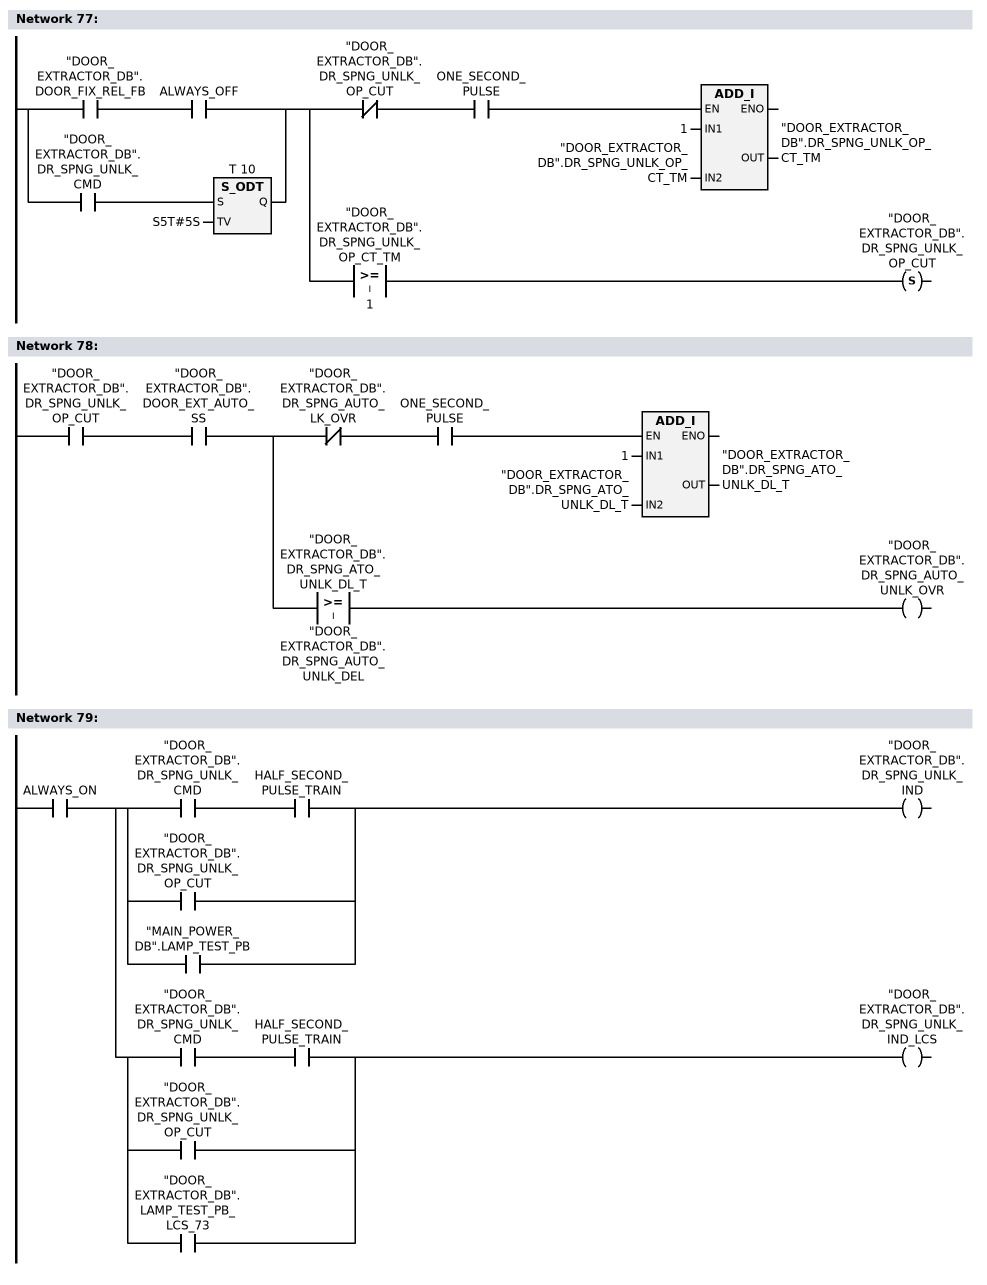
NETWORK
TITLE =
      A     "DOOR_EXTRACTOR_DB".DOOR_FIX_REL_FB;
      A     "ALWAYS_OFF";
      O(;
      A     "DOOR_EXTRACTOR_DB".DR_SPNG_UNLK_CMD;
      L     S5T#5S;
      SD    T 10;
      NOP   0;
      NOP   0;
      NOP   0;
      A     T 10;
      );
      =     L 0.0;
      A     L 0.0;
      AN    "DOOR_EXTRACTOR_DB".DR_SPNG_UNLK_OP_CUT;
      A     "ONE_SECOND_PULSE";
      JNB   M069;
      L     1;
      L     "DOOR_EXTRACTOR_DB".DR_SPNG_UNLK_OP_CT_TM;
      +I;
      T     "DOOR_EXTRACTOR_DB".DR_SPNG_UNLK_OP_CT_TM;
M069: NOP   0;
      A     L 0.0;
      A(;
      L     "DOOR_EXTRACTOR_DB".DR_SPNG_UNLK_OP_CT_TM;
      L     1;
      >=I;
      );
      S     "DOOR_EXTRACTOR_DB".DR_SPNG_UNLK_OP_CUT;
NETWORK
TITLE =
      A     "DOOR_EXTRACTOR_DB".DR_SPNG_UNLK_OP_CUT;
      A     "DOOR_EXTRACTOR_DB".DOOR_EXT_AUTO_SS;
      =     L 0.0;
      A     L 0.0;
      AN    "DOOR_EXTRACTOR_DB".DR_SPNG_AUTO_LK_OVR;
      A     "ONE_SECOND_PULSE";
      JNB   M070;
      L     1;
      L     "DOOR_EXTRACTOR_DB".DR_SPNG_ATO_UNLK_DL_T;
      +I;
      T     "DOOR_EXTRACTOR_DB".DR_SPNG_ATO_UNLK_DL_T;
M070: NOP   0;
      A     L 0.0;
      A(;
      L     "DOOR_EXTRACTOR_DB".DR_SPNG_ATO_UNLK_DL_T;
      L     "DOOR_EXTRACTOR_DB".DR_SPNG_AUTO_UNLK_DEL;
      >=I;
      );
      =     "DOOR_EXTRACTOR_DB".DR_SPNG_AUTO_UNLK_OVR;
NETWORK
TITLE =
      A     "ALWAYS_ON";
      =     L 0.0;
      A     L 0.0;
      A(;
      A     "DOOR_EXTRACTOR_DB".DR_SPNG_UNLK_CMD;
      A     "HALF_SECOND_PULSE_TRAIN";
      O     "DOOR_EXTRACTOR_DB".DR_SPNG_UNLK_OP_CUT;
      O     "MAIN_POWER_DB".LAMP_TEST_PB;
      );
      =     "DOOR_EXTRACTOR_DB".DR_SPNG_UNLK_IND;
      A     L 0.0;
      A(;
      A     "DOOR_EXTRACTOR_DB".DR_SPNG_UNLK_CMD;
      A     "HALF_SECOND_PULSE_TRAIN";
      O     "DOOR_EXTRACTOR_DB".DR_SPNG_UNLK_OP_CUT;
      O     "DOOR_EXTRACTOR_DB".LAMP_TEST_PB_LCS_73;
      );
      =     "DOOR_EXTRACTOR_DB".DR_SPNG_UNLK_IND_LCS;
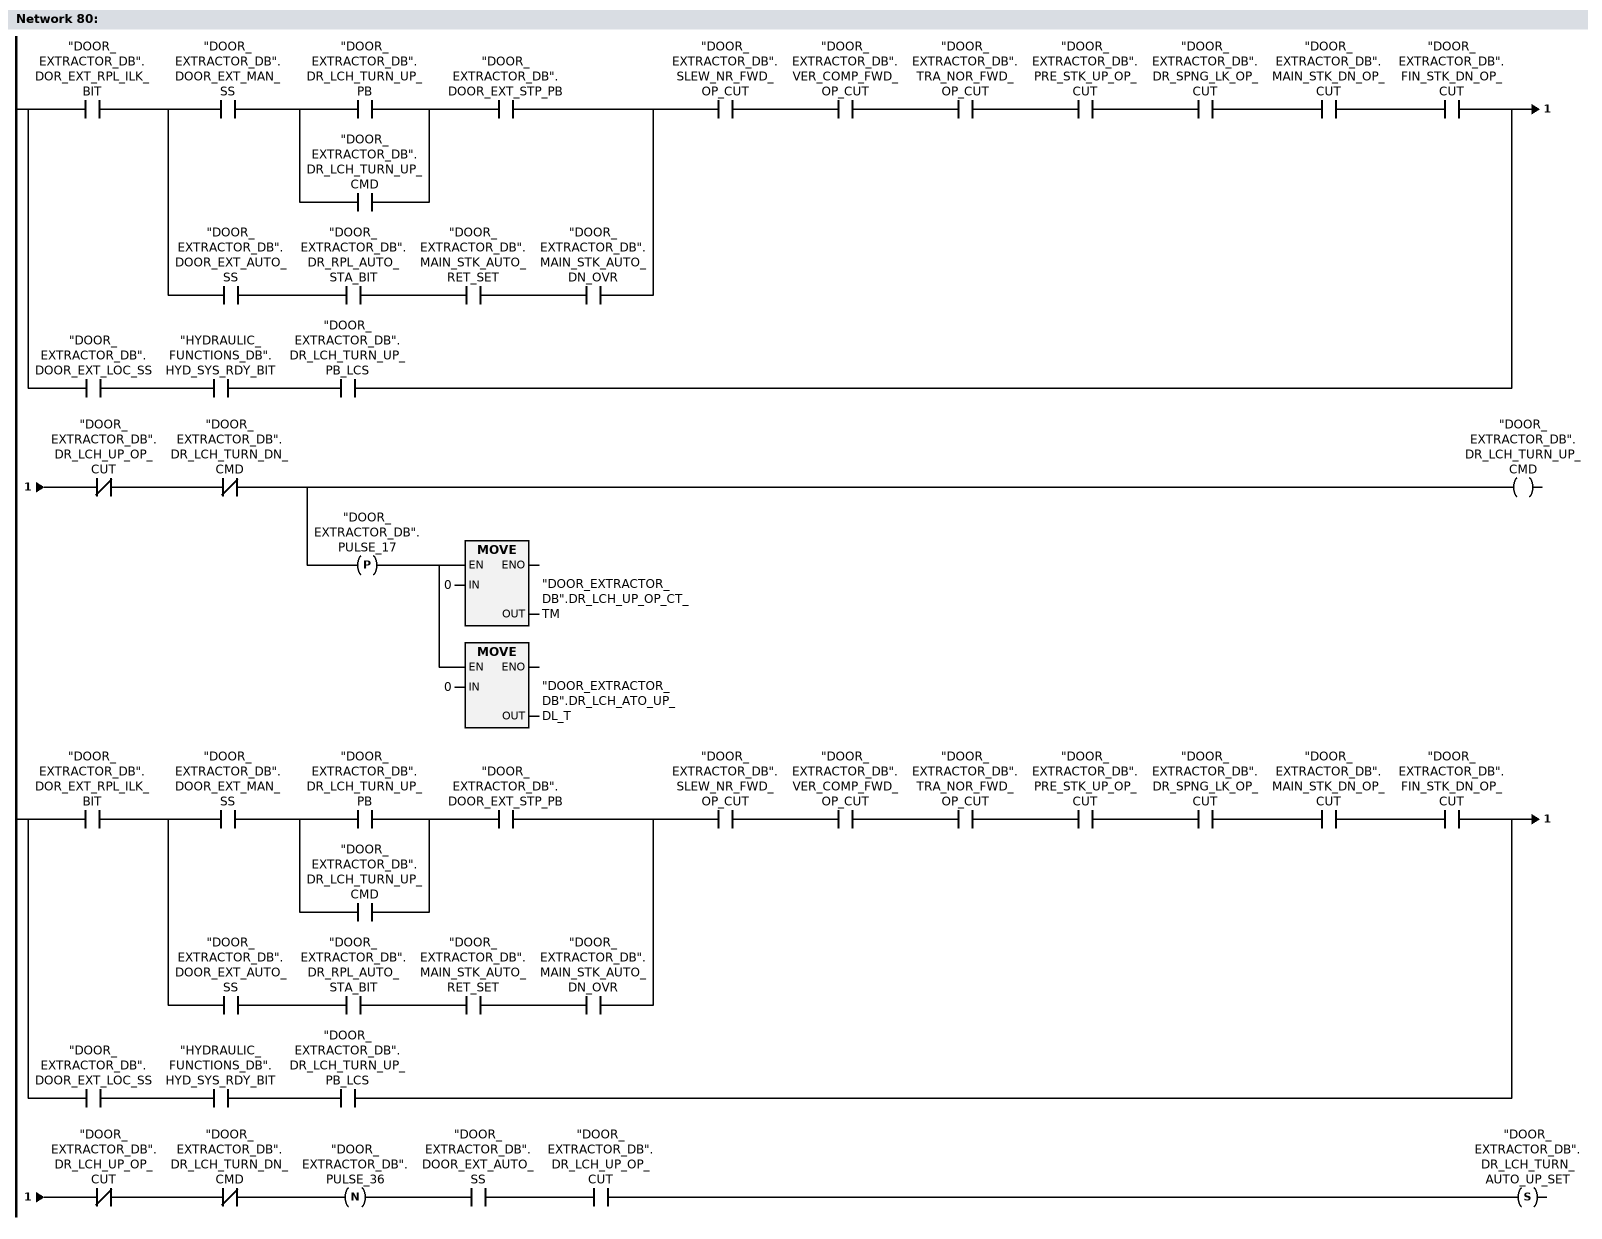
NETWORK
TITLE =
      A(;
      A     "DOOR_EXTRACTOR_DB".DOR_EXT_RPL_ILK_BIT;
      A(;
      A     "DOOR_EXTRACTOR_DB".DOOR_EXT_MAN_SS;
      A(;
      O     "DOOR_EXTRACTOR_DB".DR_LCH_TURN_UP_PB;
      O     "DOOR_EXTRACTOR_DB".DR_LCH_TURN_UP_CMD;
      );
      A     "DOOR_EXTRACTOR_DB".DOOR_EXT_STP_PB;
      O;
      A     "DOOR_EXTRACTOR_DB".DOOR_EXT_AUTO_SS;
      A     "DOOR_EXTRACTOR_DB".DR_RPL_AUTO_STA_BIT;
      A     "DOOR_EXTRACTOR_DB".MAIN_STK_AUTO_RET_SET;
      A     "DOOR_EXTRACTOR_DB".MAIN_STK_AUTO_DN_OVR;
      );
      A     "DOOR_EXTRACTOR_DB".SLEW_NR_FWD_OP_CUT;
      A     "DOOR_EXTRACTOR_DB".VER_COMP_FWD_OP_CUT;
      A     "DOOR_EXTRACTOR_DB".TRA_NOR_FWD_OP_CUT;
      A     "DOOR_EXTRACTOR_DB".PRE_STK_UP_OP_CUT;
      A     "DOOR_EXTRACTOR_DB".DR_SPNG_LK_OP_CUT;
      A     "DOOR_EXTRACTOR_DB".MAIN_STK_DN_OP_CUT;
      A     "DOOR_EXTRACTOR_DB".FIN_STK_DN_OP_CUT;
      O;
      A     "DOOR_EXTRACTOR_DB".DOOR_EXT_LOC_SS;
      A     "HYDRAULIC_FUNCTIONS_DB".HYD_SYS_RDY_BIT;
      A     "DOOR_EXTRACTOR_DB".DR_LCH_TURN_UP_PB_LCS;
      );
      AN    "DOOR_EXTRACTOR_DB".DR_LCH_UP_OP_CUT;
      AN    "DOOR_EXTRACTOR_DB".DR_LCH_TURN_DN_CMD;
      =     L 0.0;
      A     L 0.0;
      BLD   102;
      =     "DOOR_EXTRACTOR_DB".DR_LCH_TURN_UP_CMD;
      A(;
      A     L 0.0;
      FN    "DOOR_EXTRACTOR_DB".PULSE_36;
      );
      A     "DOOR_EXTRACTOR_DB".DOOR_EXT_AUTO_SS;
      A     "DOOR_EXTRACTOR_DB".DR_LCH_UP_OP_CUT;
      S     "DOOR_EXTRACTOR_DB".DR_LCH_TURN_AUTO_UP_SET;
      A     L 0.0;
      FP    "DOOR_EXTRACTOR_DB".PULSE_17;
      =     L 0.1;
      A     L 0.1;
      JNB   M071;
      L     0;
      T     "DOOR_EXTRACTOR_DB".DR_LCH_UP_OP_CT_TM;
M071: NOP   0;
      A     L 0.1;
      JNB   M072;
      L     0;
      T     "DOOR_EXTRACTOR_DB".DR_LCH_ATO_UP_DL_T;
M072: NOP   0;
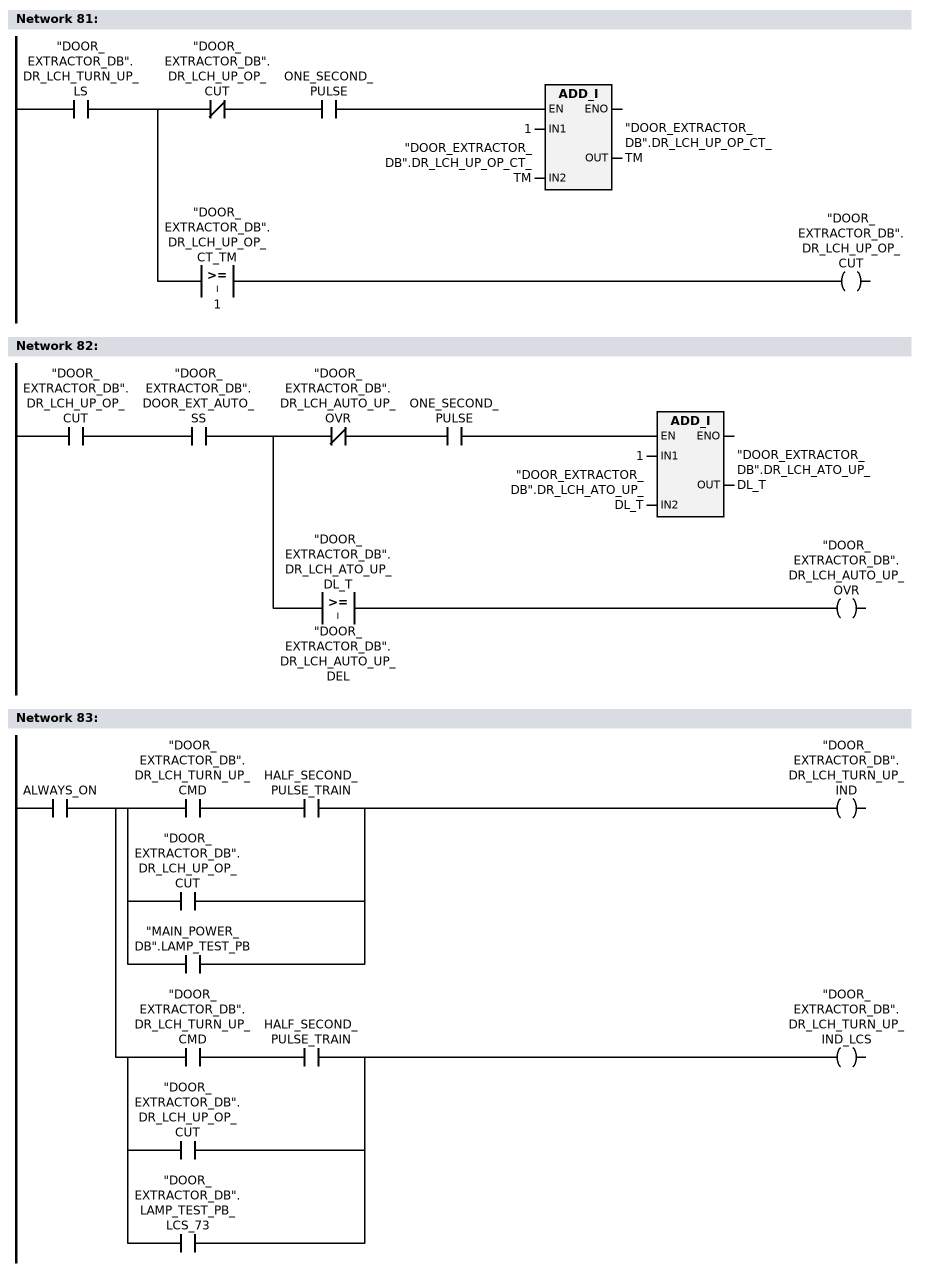
NETWORK
TITLE =
      A     "DOOR_EXTRACTOR_DB".DR_LCH_TURN_UP_LS;
      =     L 0.0;
      A     L 0.0;
      AN    "DOOR_EXTRACTOR_DB".DR_LCH_UP_OP_CUT;
      A     "ONE_SECOND_PULSE";
      JNB   M073;
      L     1;
      L     "DOOR_EXTRACTOR_DB".DR_LCH_UP_OP_CT_TM;
      +I;
      T     "DOOR_EXTRACTOR_DB".DR_LCH_UP_OP_CT_TM;
M073: NOP   0;
      A     L 0.0;
      A(;
      L     "DOOR_EXTRACTOR_DB".DR_LCH_UP_OP_CT_TM;
      L     1;
      >=I;
      );
      =     "DOOR_EXTRACTOR_DB".DR_LCH_UP_OP_CUT;
NETWORK
TITLE =
      A     "DOOR_EXTRACTOR_DB".DR_LCH_UP_OP_CUT;
      A     "DOOR_EXTRACTOR_DB".DOOR_EXT_AUTO_SS;
      =     L 0.0;
      A     L 0.0;
      AN    "DOOR_EXTRACTOR_DB".DR_LCH_AUTO_UP_OVR;
      A     "ONE_SECOND_PULSE";
      JNB   M074;
      L     1;
      L     "DOOR_EXTRACTOR_DB".DR_LCH_ATO_UP_DL_T;
      +I;
      T     "DOOR_EXTRACTOR_DB".DR_LCH_ATO_UP_DL_T;
M074: NOP   0;
      A     L 0.0;
      A(;
      L     "DOOR_EXTRACTOR_DB".DR_LCH_ATO_UP_DL_T;
      L     "DOOR_EXTRACTOR_DB".DR_LCH_AUTO_UP_DEL;
      >=I;
      );
      =     "DOOR_EXTRACTOR_DB".DR_LCH_AUTO_UP_OVR;
NETWORK
TITLE =
      A     "ALWAYS_ON";
      =     L 0.0;
      A     L 0.0;
      A(;
      A     "DOOR_EXTRACTOR_DB".DR_LCH_TURN_UP_CMD;
      A     "HALF_SECOND_PULSE_TRAIN";
      O     "DOOR_EXTRACTOR_DB".DR_LCH_UP_OP_CUT;
      O     "MAIN_POWER_DB".LAMP_TEST_PB;
      );
      =     "DOOR_EXTRACTOR_DB".DR_LCH_TURN_UP_IND;
      A     L 0.0;
      A(;
      A     "DOOR_EXTRACTOR_DB".DR_LCH_TURN_UP_CMD;
      A     "HALF_SECOND_PULSE_TRAIN";
      O     "DOOR_EXTRACTOR_DB".DR_LCH_UP_OP_CUT;
      O     "DOOR_EXTRACTOR_DB".LAMP_TEST_PB_LCS_73;
      );
      =     "DOOR_EXTRACTOR_DB".DR_LCH_TURN_UP_IND_LCS;
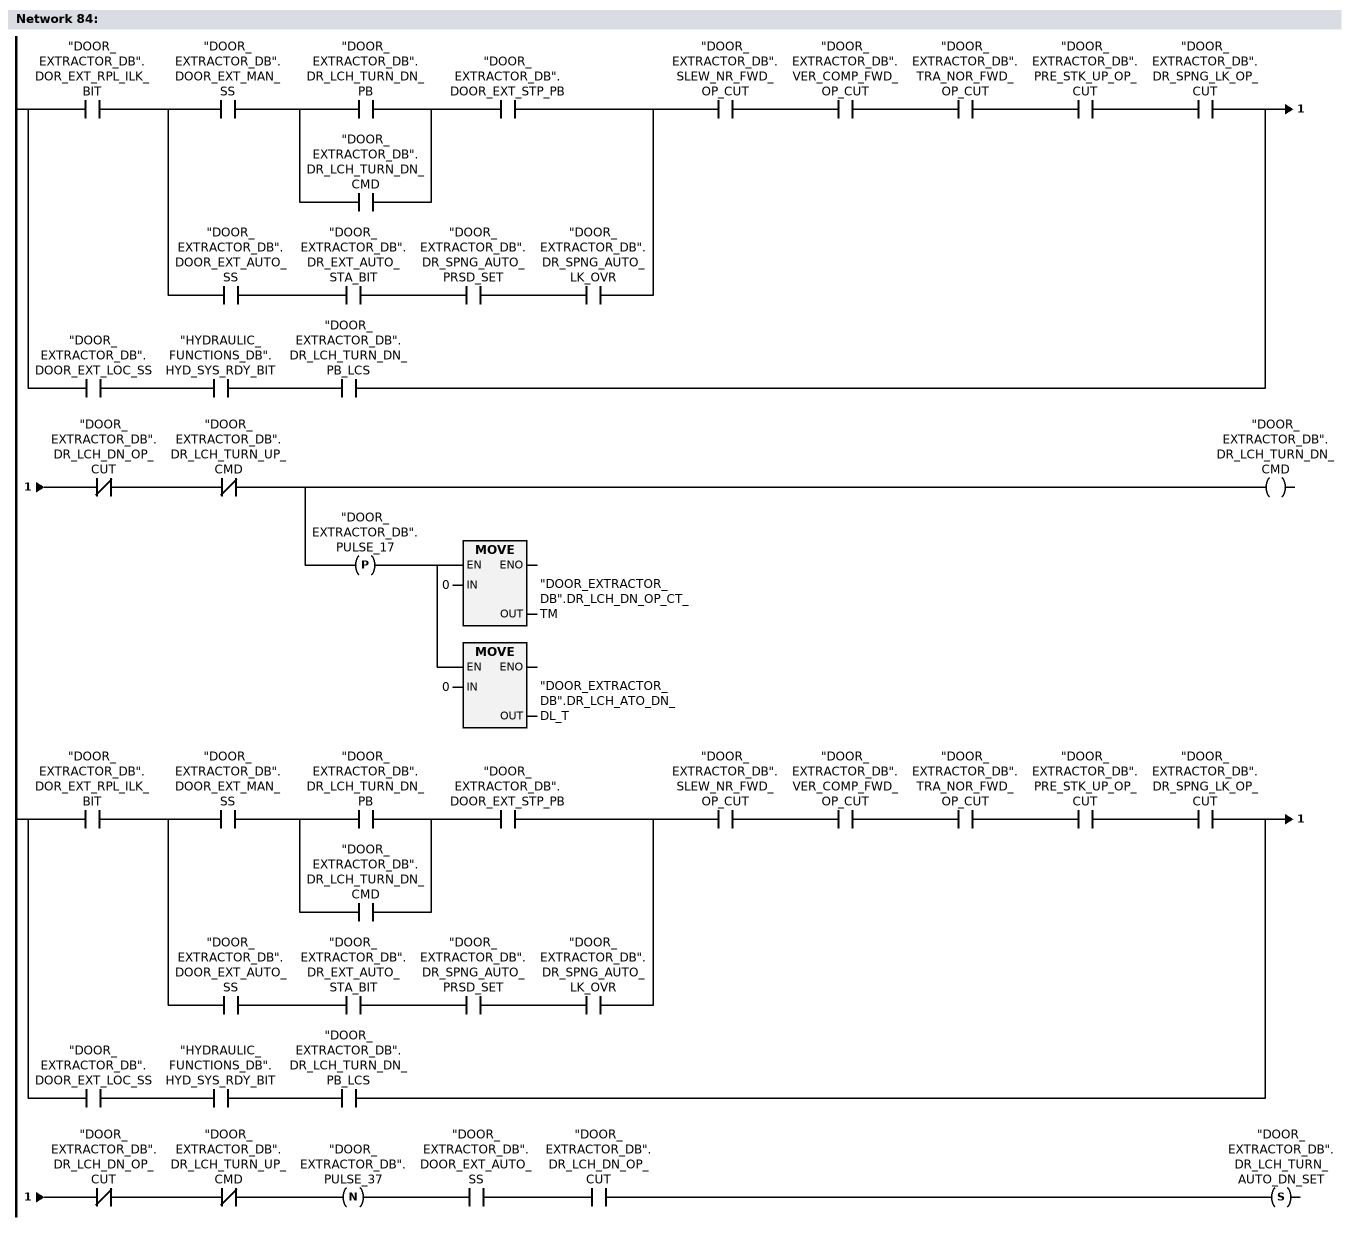
NETWORK
TITLE =
      A(;
      A     "DOOR_EXTRACTOR_DB".DOR_EXT_RPL_ILK_BIT;
      A(;
      A     "DOOR_EXTRACTOR_DB".DOOR_EXT_MAN_SS;
      A(;
      O     "DOOR_EXTRACTOR_DB".DR_LCH_TURN_DN_PB;
      O     "DOOR_EXTRACTOR_DB".DR_LCH_TURN_DN_CMD;
      );
      A     "DOOR_EXTRACTOR_DB".DOOR_EXT_STP_PB;
      O;
      A     "DOOR_EXTRACTOR_DB".DOOR_EXT_AUTO_SS;
      A     "DOOR_EXTRACTOR_DB".DR_EXT_AUTO_STA_BIT;
      A     "DOOR_EXTRACTOR_DB".DR_SPNG_AUTO_PRSD_SET;
      A     "DOOR_EXTRACTOR_DB".DR_SPNG_AUTO_LK_OVR;
      );
      A     "DOOR_EXTRACTOR_DB".SLEW_NR_FWD_OP_CUT;
      A     "DOOR_EXTRACTOR_DB".VER_COMP_FWD_OP_CUT;
      A     "DOOR_EXTRACTOR_DB".TRA_NOR_FWD_OP_CUT;
      A     "DOOR_EXTRACTOR_DB".PRE_STK_UP_OP_CUT;
      A     "DOOR_EXTRACTOR_DB".DR_SPNG_LK_OP_CUT;
      O;
      A     "DOOR_EXTRACTOR_DB".DOOR_EXT_LOC_SS;
      A     "HYDRAULIC_FUNCTIONS_DB".HYD_SYS_RDY_BIT;
      A     "DOOR_EXTRACTOR_DB".DR_LCH_TURN_DN_PB_LCS;
      );
      AN    "DOOR_EXTRACTOR_DB".DR_LCH_DN_OP_CUT;
      AN    "DOOR_EXTRACTOR_DB".DR_LCH_TURN_UP_CMD;
      =     L 0.0;
      A     L 0.0;
      BLD   102;
      =     "DOOR_EXTRACTOR_DB".DR_LCH_TURN_DN_CMD;
      A(;
      A     L 0.0;
      FN    "DOOR_EXTRACTOR_DB".PULSE_37;
      );
      A     "DOOR_EXTRACTOR_DB".DOOR_EXT_AUTO_SS;
      A     "DOOR_EXTRACTOR_DB".DR_LCH_DN_OP_CUT;
      S     "DOOR_EXTRACTOR_DB".DR_LCH_TURN_AUTO_DN_SET;
      A     L 0.0;
      FP    "DOOR_EXTRACTOR_DB".PULSE_17;
      =     L 0.1;
      A     L 0.1;
      JNB   M075;
      L     0;
      T     "DOOR_EXTRACTOR_DB".DR_LCH_DN_OP_CT_TM;
M075: NOP   0;
      A     L 0.1;
      JNB   M076;
      L     0;
      T     "DOOR_EXTRACTOR_DB".DR_LCH_ATO_DN_DL_T;
M076: NOP   0;
